Yaskawa INFORM job: pointsclTRJ1.JBI

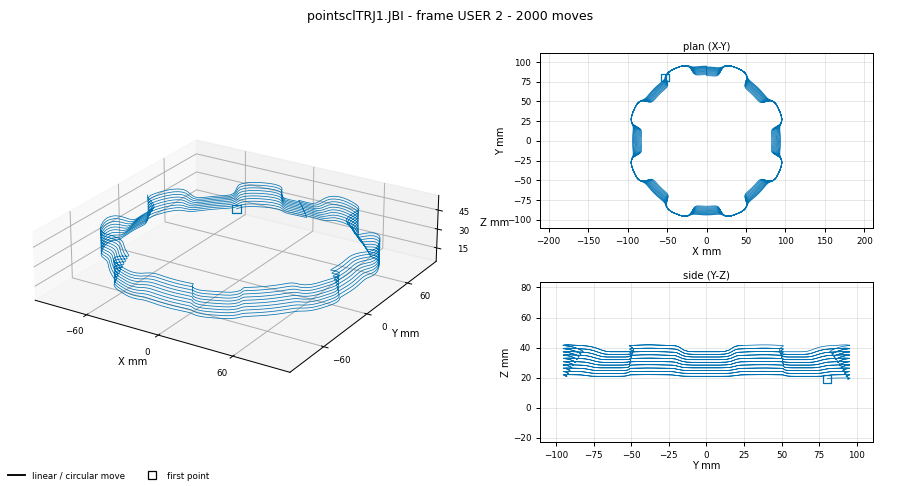
[picture p0: tool path of pointsclTRJ1.JBI in frame USER 2, 2000 of 2000 moves have a stored position in this frame; points joined in program order, loops and branches not executed]
/JOB
//NAME pointsclTRJ1
//POS
///NPOS 2000,0,0,0,0,0
///USER 2
///TOOL 1
///POSTYPE USER
///RECTAN
///RCONF 1,0,0,0,0,0,0,0,0,0,0,0,0,0,0,0,0,0,0,0,0,0,0,0
C00000=-52.755,80.388,19.309,-159.4943,21.2238,0.0000
C00001=-51.961,81.931,19.493,-161.2614,21.3884,0.0000
C00002=-51.163,83.502,19.627,-163.2617,21.3173,0.0000
C00003=-49.917,85.194,19.692,-165.6695,20.6930,0.0000
C00004=-47.874,87.106,19.726,-168.7116,19.3736,0.0000
C00005=-45.272,88.975,19.753,-171.6554,17.3027,0.0000
C00006=-42.449,90.515,19.780,-179.9091,0.0437,0.0000
C00007=-39.659,91.796,19.798,-179.9891,0.0048,0.0000
C00008=-36.867,92.953,19.798,-179.9889,0.0043,0.0000
C00009=-33.988,94.020,19.780,-179.9048,0.0334,0.0000
C00010=-30.903,94.927,19.753,-161.9258,-6.4497,0.0000
C00011=-27.741,95.446,19.726,-158.4611,-5.9689,0.0000
C00012=-24.945,95.538,19.692,-155.4722,-4.9413,0.0000
C00013=-22.867,95.222,19.627,-153.3983,-3.8614,0.0000
C00014=-21.192,94.676,19.493,-151.9726,-2.6572,0.0000
C00015=-19.540,94.146,19.309,-150.8542,-1.4373,0.0000
C00016=-17.528,93.824,19.120,-149.8453,-0.1078,0.0000
C00017=-14.592,93.857,18.976,-148.8983,1.4069,0.0000
C00018=-10.190,94.262,18.917,-148.2538,2.5071,0.0000
C00019=-5.317,94.652,18.914,-148.1214,1.7626,0.0000
C00020=0.000,94.804,18.916,-148.0939,0.0004,0.0000
C00021=0.000,93.772,20.859,-146.9132,0.0004,0.0000
C00022=5.223,93.624,20.857,-146.9416,-1.8172,0.0000
C00023=10.031,93.243,20.860,-147.0713,-2.4820,0.0000
C00024=14.399,92.874,20.935,-147.7018,-1.1471,0.0000
C00025=17.292,92.935,21.118,-148.6350,0.5162,0.0000
C00026=19.271,93.399,21.361,-149.6419,1.9341,0.0000
C00027=20.902,94.108,21.598,-150.7809,3.2271,0.0000
C00028=22.556,94.852,21.773,-152.2300,4.6103,0.0000
C00029=24.607,95.353,21.858,-154.3520,5.8653,0.0000
C00030=27.423,95.407,21.902,-157.4539,7.0484,0.0000
C00031=30.651,94.973,21.938,-161.0071,7.6664,0.0000
C00032=33.828,94.073,21.973,-164.2005,7.6094,0.0000
C00033=36.813,92.974,21.997,-179.9889,-0.0043,0.0000
C00034=39.712,91.773,21.997,-179.9891,-0.0048,0.0000
C00035=42.599,90.440,21.973,-174.1812,-16.5268,0.0000
C00036=45.483,88.829,21.938,-171.8779,-18.8083,0.0000
C00037=48.072,86.854,21.902,-168.7509,-20.8451,0.0000
C00038=50.025,84.825,21.858,-165.4828,-22.1308,0.0000
C00039=51.121,83.020,21.773,-162.8864,-22.6578,0.0000
C00040=51.765,81.324,21.598,-160.7193,-22.6085,0.0000
C00041=52.416,79.670,21.361,-158.8690,-22.3978,0.0000
C00042=53.488,77.942,21.118,-157.0442,-21.9870,0.0000
C00043=55.491,75.854,20.935,-155.1213,-21.3210,0.0000
C00044=58.840,73.026,20.860,-153.6891,-20.6953,0.0000
C00045=62.509,69.895,20.857,-154.0343,-21.2910,0.0000
C00046=66.307,66.307,20.859,-155.2636,-22.7071,0.0000
C00047=69.895,62.509,20.857,-156.5650,-24.0758,0.0000
C00048=73.026,58.840,20.860,-157.1474,-24.4962,0.0000
C00049=75.854,55.491,20.935,-156.7212,-23.0730,0.0000
C00050=77.942,53.488,21.118,-156.3234,-21.2020,0.0000
C00051=79.670,52.416,21.361,-156.1628,-19.4697,0.0000
C00052=81.324,51.765,21.598,-156.1941,-17.7476,0.0000
C00053=83.020,51.121,21.773,-156.4051,-15.7569,0.0000
C00054=84.825,50.025,21.858,-157.2128,-13.4268,0.0000
C00055=86.854,48.072,21.902,-158.7826,-10.5041,0.0000
C00056=88.829,45.483,21.938,-161.0147,-7.6857,0.0000
C00057=90.440,42.599,21.973,-163.3923,-5.5777,0.0000
C00058=91.773,39.712,21.997,-179.9952,-0.0109,0.0000
C00059=92.974,36.813,21.997,-179.9957,-0.0111,0.0000
C00060=94.073,33.828,21.973,172.0955,-15.6567,0.0000
C00061=94.973,30.651,21.938,171.8979,-18.8167,0.0000
C00062=95.407,27.423,21.902,172.3749,-22.3664,0.0000
C00063=95.353,24.607,21.858,173.4988,-25.5041,0.0000
C00064=94.852,22.556,21.773,174.7928,-27.6724,0.0000
C00065=94.108,20.902,21.598,176.3037,-29.1683,0.0000
C00066=93.399,19.271,21.361,177.7589,-30.3389,0.0000
C00067=92.935,17.292,21.118,179.3955,-31.3636,0.0000
C00068=92.874,14.399,20.935,-178.6430,-32.2909,0.0000
C00069=93.243,10.031,20.860,-177.0437,-32.8939,0.0000
C00070=93.624,5.223,20.857,-177.8321,-33.0396,0.0000
C00071=93.772,0.000,20.859,179.9995,-33.0868,0.0000
C00072=93.624,-5.223,20.857,177.8327,-33.0396,0.0000
C00073=93.243,-10.031,20.860,177.0444,-32.8939,0.0000
C00074=92.875,-14.399,20.935,178.6429,-32.2908,0.0000
C00075=92.935,-17.292,21.118,-179.3958,-31.3634,0.0000
C00076=93.399,-19.271,21.361,-177.7592,-30.3389,0.0000
C00077=94.108,-20.902,21.598,-176.3039,-29.1683,0.0000
C00078=94.852,-22.556,21.773,-174.7928,-27.6724,0.0000
C00079=95.353,-24.607,21.858,-173.4988,-25.5041,0.0000
C00080=95.407,-27.423,21.902,-172.3749,-22.3664,0.0000
C00081=94.973,-30.651,21.938,-171.8979,-18.8167,0.0000
C00082=94.073,-33.828,21.973,-172.0955,-15.6567,0.0000
C00083=92.974,-36.813,21.997,179.9957,-0.0111,0.0000
C00084=91.773,-39.712,21.997,179.9952,-0.0109,0.0000
C00085=90.440,-42.599,21.973,163.3923,-5.5777,0.0000
C00086=88.829,-45.483,21.938,161.0147,-7.6857,0.0000
C00087=86.854,-48.072,21.902,158.7826,-10.5041,0.0000
C00088=84.825,-50.025,21.858,157.2128,-13.4268,0.0000
C00089=83.020,-51.121,21.773,156.4050,-15.7569,0.0000
C00090=81.324,-51.765,21.598,156.1939,-17.7474,0.0000
C00091=79.670,-52.416,21.361,156.1625,-19.4695,0.0000
C00092=77.942,-53.488,21.118,156.3231,-21.2019,0.0000
C00093=75.854,-55.491,20.935,156.7211,-23.0731,0.0000
C00094=73.026,-58.840,20.860,157.1478,-24.4967,0.0000
C00095=69.895,-62.509,20.857,156.5653,-24.0762,0.0000
C00096=66.307,-66.307,20.859,155.2630,-22.7065,0.0000
C00097=62.509,-69.895,20.857,154.0346,-21.2914,0.0000
C00098=58.840,-73.026,20.860,153.6895,-20.6957,0.0000
C00099=55.491,-75.854,20.935,155.1214,-21.3209,0.0000
C00100=53.488,-77.942,21.118,157.0440,-21.9867,0.0000
C00101=52.416,-79.670,21.361,158.8689,-22.3975,0.0000
C00102=51.765,-81.324,21.598,160.7192,-22.6084,0.0000
C00103=51.121,-83.020,21.773,162.8864,-22.6578,0.0000
C00104=50.025,-84.825,21.858,165.4828,-22.1308,0.0000
C00105=48.072,-86.854,21.902,168.7509,-20.8451,0.0000
C00106=45.483,-88.829,21.938,171.8779,-18.8083,0.0000
C00107=42.599,-90.440,21.973,174.1812,-16.5268,0.0000
C00108=39.712,-91.773,21.997,179.9891,-0.0048,0.0000
C00109=36.813,-92.974,21.997,179.9889,-0.0043,0.0000
C00110=33.828,-94.073,21.973,164.2005,7.6094,0.0000
C00111=30.651,-94.973,21.938,161.0071,7.6664,0.0000
C00112=27.423,-95.407,21.902,157.4539,7.0484,0.0000
C00113=24.607,-95.353,21.858,154.3520,5.8653,0.0000
C00114=22.556,-94.852,21.773,152.2300,4.6103,0.0000
C00115=20.902,-94.108,21.598,150.7809,3.2271,0.0000
C00116=19.271,-93.399,21.361,149.6419,1.9341,0.0000
C00117=17.292,-92.935,21.118,148.6350,0.5162,0.0000
C00118=14.399,-92.874,20.935,147.7018,-1.1471,0.0000
C00119=10.031,-93.243,20.860,147.0713,-2.4820,0.0000
C00120=5.223,-93.624,20.857,146.9416,-1.8172,0.0000
C00121=0.000,-93.772,20.859,146.9132,0.0004,0.0000
C00122=0.000,-93.772,20.859,146.9132,0.0004,0.0000
C00123=-5.223,-93.624,20.857,146.9416,1.8167,0.0000
C00124=-10.031,-93.243,20.860,147.0713,2.4814,0.0000
C00125=-14.399,-92.875,20.935,147.7020,1.1472,0.0000
C00126=-17.292,-92.935,21.118,148.6351,-0.5159,0.0000
C00127=-19.271,-93.399,21.361,149.6420,-1.9338,0.0000
C00128=-20.902,-94.108,21.598,150.7809,-3.2269,0.0000
C00129=-22.556,-94.852,21.773,152.2300,-4.6102,0.0000
C00130=-24.607,-95.353,21.858,154.3520,-5.8653,0.0000
C00131=-27.423,-95.407,21.902,157.4539,-7.0484,0.0000
C00132=-30.651,-94.973,21.938,161.0071,-7.6664,0.0000
C00133=-33.828,-94.073,21.973,164.2005,-7.6094,0.0000
C00134=-36.813,-92.974,21.997,179.9889,0.0043,0.0000
C00135=-39.712,-91.773,21.997,179.9891,0.0048,0.0000
C00136=-42.599,-90.440,21.973,174.1812,16.5268,0.0000
C00137=-45.483,-88.829,21.938,171.8779,18.8083,0.0000
C00138=-48.072,-86.854,21.902,168.7509,20.8451,0.0000
C00139=-50.025,-84.825,21.858,165.4828,22.1308,0.0000
C00140=-51.121,-83.020,21.773,162.8864,22.6578,0.0000
C00141=-51.765,-81.324,21.598,160.7193,22.6085,0.0000
C00142=-52.416,-79.670,21.361,158.8690,22.3978,0.0000
C00143=-53.488,-77.942,21.118,157.0442,21.9870,0.0000
C00144=-55.491,-75.854,20.935,155.1213,21.3210,0.0000
C00145=-58.840,-73.026,20.860,153.6891,20.6953,0.0000
C00146=-62.509,-69.895,20.857,154.0343,21.2910,0.0000
C00147=-66.307,-66.307,20.859,155.2636,22.7071,0.0000
C00148=-69.895,-62.509,20.857,156.5650,24.0758,0.0000
C00149=-73.026,-58.840,20.860,157.1474,24.4962,0.0000
C00150=-75.854,-55.491,20.935,156.7212,23.0730,0.0000
C00151=-77.942,-53.488,21.118,156.3234,21.2020,0.0000
C00152=-79.670,-52.416,21.361,156.1628,19.4697,0.0000
C00153=-81.324,-51.765,21.598,156.1941,17.7476,0.0000
C00154=-83.020,-51.121,21.773,156.4051,15.7569,0.0000
C00155=-84.825,-50.025,21.858,157.2128,13.4268,0.0000
C00156=-86.854,-48.072,21.902,158.7826,10.5041,0.0000
C00157=-88.829,-45.483,21.938,161.0147,7.6857,0.0000
C00158=-90.440,-42.599,21.973,163.3923,5.5777,0.0000
C00159=-91.773,-39.712,21.997,179.9952,0.0109,0.0000
C00160=-92.974,-36.813,21.997,179.9957,0.0111,0.0000
C00161=-94.073,-33.828,21.973,-172.0955,15.6567,0.0000
C00162=-94.973,-30.651,21.938,-171.8979,18.8167,0.0000
C00163=-95.407,-27.423,21.902,-172.3749,22.3664,0.0000
C00164=-95.353,-24.607,21.858,-173.4988,25.5041,0.0000
C00165=-94.852,-22.556,21.773,-174.7928,27.6724,0.0000
C00166=-94.108,-20.902,21.598,-176.3037,29.1683,0.0000
C00167=-93.399,-19.271,21.361,-177.7589,30.3389,0.0000
C00168=-92.935,-17.292,21.118,-179.3955,31.3636,0.0000
C00169=-92.874,-14.399,20.935,178.6430,32.2909,0.0000
C00170=-93.243,-10.031,20.860,177.0437,32.8939,0.0000
C00171=-93.624,-5.223,20.857,177.8321,33.0396,0.0000
C00172=-93.772,0.000,20.859,-179.9995,33.0868,0.0000
C00173=-93.624,5.223,20.857,-177.8327,33.0396,0.0000
C00174=-93.243,10.031,20.860,-177.0444,32.8939,0.0000
C00175=-92.875,14.399,20.935,-178.6429,32.2908,0.0000
C00176=-92.935,17.292,21.118,179.3958,31.3634,0.0000
C00177=-93.399,19.271,21.361,177.7592,30.3389,0.0000
C00178=-94.108,20.902,21.598,176.3039,29.1683,0.0000
C00179=-94.852,22.556,21.773,174.7928,27.6724,0.0000
C00180=-95.353,24.607,21.858,173.4988,25.5041,0.0000
C00181=-95.407,27.423,21.902,172.3749,22.3664,0.0000
C00182=-94.973,30.651,21.938,171.8979,18.8167,0.0000
C00183=-94.073,33.828,21.973,172.0955,15.6567,0.0000
C00184=-92.974,36.813,21.997,-179.9957,0.0111,0.0000
C00185=-91.773,39.712,21.997,-179.9952,0.0109,0.0000
C00186=-90.440,42.599,21.973,-163.3923,5.5777,0.0000
C00187=-88.829,45.483,21.938,-161.0147,7.6857,0.0000
C00188=-86.854,48.072,21.902,-158.7826,10.5041,0.0000
C00189=-84.825,50.025,21.858,-157.2128,13.4268,0.0000
C00190=-83.020,51.121,21.773,-156.4050,15.7569,0.0000
C00191=-81.324,51.765,21.598,-156.1939,17.7474,0.0000
C00192=-79.670,52.416,21.361,-156.1625,19.4695,0.0000
C00193=-77.942,53.488,21.118,-156.3231,21.2019,0.0000
C00194=-75.854,55.491,20.935,-156.7211,23.0731,0.0000
C00195=-73.026,58.840,20.860,-157.1478,24.4967,0.0000
C00196=-69.895,62.509,20.857,-156.5653,24.0762,0.0000
C00197=-66.307,66.307,20.859,-155.2630,22.7065,0.0000
C00198=-62.509,69.895,20.857,-154.0346,21.2914,0.0000
C00199=-58.840,73.026,20.860,-153.6895,20.6957,0.0000
C00200=-55.491,75.854,20.935,-155.1214,21.3209,0.0000
C00201=-53.488,77.942,21.118,-157.0440,21.9867,0.0000
C00202=-52.416,79.670,21.361,-158.8689,22.3975,0.0000
C00203=-51.765,81.324,21.598,-160.7192,22.6084,0.0000
C00204=-51.121,83.020,21.773,-162.8864,22.6578,0.0000
C00205=-50.025,84.825,21.858,-165.4828,22.1308,0.0000
C00206=-48.072,86.854,21.902,-168.7509,20.8451,0.0000
C00207=-45.483,88.829,21.938,-171.8779,18.8083,0.0000
C00208=-42.599,90.440,21.973,-174.1812,16.5268,0.0000
C00209=-39.712,91.773,21.997,-179.9891,0.0048,0.0000
C00210=-36.813,92.974,21.997,-179.9889,0.0043,0.0000
C00211=-33.828,94.073,21.973,-164.2005,-7.6094,0.0000
C00212=-30.651,94.973,21.938,-161.0071,-7.6664,0.0000
C00213=-27.423,95.407,21.902,-157.4539,-7.0484,0.0000
C00214=-24.607,95.353,21.858,-154.3520,-5.8653,0.0000
C00215=-22.556,94.852,21.773,-152.2300,-4.6102,0.0000
C00216=-20.902,94.108,21.598,-150.7809,-3.2269,0.0000
C00217=-19.271,93.399,21.361,-149.6420,-1.9338,0.0000
C00218=-17.292,92.935,21.118,-148.6351,-0.5159,0.0000
C00219=-14.399,92.875,20.935,-147.7020,1.1472,0.0000
C00220=-10.031,93.243,20.860,-147.0713,2.4814,0.0000
C00221=-5.223,93.624,20.857,-146.9416,1.8167,0.0000
C00222=0.000,93.772,20.859,-146.9132,0.0004,0.0000
C00223=0.000,92.684,22.771,-145.8888,0.0004,0.0000
C00224=5.124,92.540,22.769,-145.9181,-1.8620,0.0000
C00225=9.864,92.169,22.773,-146.0452,-2.4396,0.0000
C00226=14.194,91.838,22.865,-146.6687,-0.8798,0.0000
C00227=17.042,91.994,23.091,-147.5969,0.9153,0.0000
C00228=18.986,92.606,23.393,-148.6082,2.4100,0.0000
C00229=20.592,93.503,23.691,-149.7732,3.7684,0.0000
C00230=22.223,94.456,23.912,-151.2813,5.2238,0.0000
C00231=24.245,95.156,24.019,-153.4766,6.7389,0.0000
C00232=27.082,95.366,24.075,-156.7610,8.0545,0.0000
C00233=30.380,95.022,24.120,-160.5087,8.7471,0.0000
C00234=33.658,94.129,24.166,-163.7677,8.7396,0.0000
C00235=36.755,92.996,24.196,-179.9893,-0.0042,0.0000
C00236=39.769,91.748,24.196,-179.9895,-0.0046,0.0000
C00237=42.760,90.359,24.166,-174.7067,-17.6262,0.0000
C00238=45.709,88.673,24.120,-172.3190,-19.9210,0.0000
C00239=48.284,86.584,24.075,-168.9803,-22.0444,0.0000
C00240=50.142,84.429,24.019,-165.4510,-23.3634,0.0000
C00241=51.076,82.504,23.912,-162.5826,-23.7496,0.0000
C00242=51.556,80.678,23.691,-160.2983,-23.6832,0.0000
C00243=52.057,78.907,23.393,-158.3658,-23.4364,0.0000
C00244=52.999,77.101,23.091,-156.4709,-22.9648,0.0000
C00245=54.903,74.976,22.865,-154.4508,-22.1874,0.0000
C00246=58.198,72.148,22.773,-152.8667,-21.3762,0.0000
C00247=61.813,69.059,22.769,-153.1525,-21.9046,0.0000
C00248=65.538,65.538,22.771,-154.4083,-23.3627,0.0000
C00249=69.059,61.813,22.769,-155.7401,-24.7719,0.0000
C00250=72.148,58.198,22.773,-156.2588,-25.1304,0.0000
C00251=74.976,54.903,22.865,-155.6753,-23.5376,0.0000
C00252=77.101,52.999,23.091,-155.1950,-21.5663,0.0000
C00253=78.907,52.057,23.393,-154.9986,-19.7713,0.0000
C00254=80.678,51.556,23.691,-155.0197,-17.9829,0.0000
C00255=82.504,51.076,23.912,-155.2435,-15.9014,0.0000
C00256=84.429,50.142,24.019,-155.9492,-13.3330,0.0000
C00257=86.584,48.284,24.075,-157.5822,-10.2051,0.0000
C00258=88.673,45.709,24.120,-159.9130,-7.2188,0.0000
C00259=90.359,42.760,24.166,-162.3030,-5.0442,0.0000
C00260=91.748,39.769,24.196,-179.9954,-0.0105,0.0000
C00261=92.996,36.755,24.196,-179.9958,-0.0107,0.0000
C00262=94.129,33.658,24.166,170.9035,-16.0387,0.0000
C00263=95.022,30.380,24.120,170.7301,-19.2556,0.0000
C00264=95.366,27.082,24.075,171.2449,-22.9965,0.0000
C00265=95.156,24.245,24.019,172.4771,-26.3260,0.0000
C00266=94.456,22.223,23.912,174.0484,-28.5884,0.0000
C00267=93.503,20.592,23.691,175.6407,-30.1546,0.0000
C00268=92.606,18.986,23.393,177.1774,-31.3609,0.0000
C00269=91.994,17.042,23.091,178.9159,-32.3984,0.0000
C00270=91.838,14.194,22.865,-178.9471,-33.3268,0.0000
C00271=92.169,9.864,22.773,-177.0596,-33.9199,0.0000
C00272=92.540,5.124,22.769,-177.7522,-34.0614,0.0000
C00273=92.684,0.000,22.771,179.9995,-34.1112,0.0000
C00274=92.540,-5.124,22.769,177.7528,-34.0615,0.0000
C00275=92.169,-9.864,22.773,177.0604,-33.9198,0.0000
C00276=91.838,-14.194,22.865,178.9470,-33.3267,0.0000
C00277=91.994,-17.042,23.091,-178.9163,-32.3983,0.0000
C00278=92.606,-18.986,23.393,-177.1778,-31.3608,0.0000
C00279=93.503,-20.592,23.691,-175.6410,-30.1546,0.0000
C00280=94.456,-22.223,23.912,-174.0485,-28.5884,0.0000
C00281=95.156,-24.245,24.019,-172.4771,-26.3260,0.0000
C00282=95.366,-27.082,24.075,-171.2449,-22.9965,0.0000
C00283=95.022,-30.380,24.120,-170.7301,-19.2556,0.0000
C00284=94.129,-33.658,24.166,-170.9035,-16.0387,0.0000
C00285=92.996,-36.755,24.196,179.9958,-0.0107,0.0000
C00286=91.748,-39.769,24.196,179.9954,-0.0105,0.0000
C00287=90.359,-42.760,24.166,162.3030,-5.0442,0.0000
C00288=88.673,-45.709,24.120,159.9130,-7.2188,0.0000
C00289=86.584,-48.284,24.075,157.5822,-10.2051,0.0000
C00290=84.429,-50.142,24.019,155.9492,-13.3330,0.0000
C00291=82.504,-51.076,23.912,155.2435,-15.9013,0.0000
C00292=80.678,-51.556,23.691,155.0196,-17.9828,0.0000
C00293=78.907,-52.057,23.393,154.9983,-19.7711,0.0000
C00294=77.101,-52.999,23.091,155.1947,-21.5661,0.0000
C00295=74.976,-54.903,22.865,155.6752,-23.5376,0.0000
C00296=72.148,-58.198,22.773,156.2592,-25.1309,0.0000
C00297=69.059,-61.813,22.769,155.7405,-24.7723,0.0000
C00298=65.538,-65.538,22.771,154.4077,-23.3621,0.0000
C00299=61.813,-69.059,22.769,153.1528,-21.9050,0.0000
C00300=58.198,-72.148,22.773,152.8672,-21.3767,0.0000
C00301=54.903,-74.976,22.865,154.4508,-22.1873,0.0000
C00302=52.999,-77.101,23.091,156.4708,-22.9645,0.0000
C00303=52.057,-78.907,23.393,158.3656,-23.4361,0.0000
C00304=51.556,-80.678,23.691,160.2982,-23.6830,0.0000
C00305=51.076,-82.504,23.912,162.5826,-23.7495,0.0000
C00306=50.142,-84.429,24.019,165.4510,-23.3634,0.0000
C00307=48.284,-86.584,24.075,168.9803,-22.0444,0.0000
C00308=45.709,-88.673,24.120,172.3190,-19.9210,0.0000
C00309=42.760,-90.359,24.166,174.7067,-17.6262,0.0000
C00310=39.769,-91.748,24.196,179.9895,-0.0046,0.0000
C00311=36.755,-92.996,24.196,179.9893,-0.0042,0.0000
C00312=33.658,-94.129,24.166,163.7677,8.7396,0.0000
C00313=30.380,-95.022,24.120,160.5087,8.7471,0.0000
C00314=27.082,-95.366,24.075,156.7610,8.0545,0.0000
C00315=24.245,-95.156,24.019,153.4766,6.7389,0.0000
C00316=22.223,-94.456,23.912,151.2813,5.2238,0.0000
C00317=20.592,-93.503,23.691,149.7732,3.7684,0.0000
C00318=18.986,-92.606,23.393,148.6082,2.4100,0.0000
C00319=17.042,-91.994,23.091,147.5969,0.9153,0.0000
C00320=14.194,-91.838,22.865,146.6687,-0.8798,0.0000
C00321=9.864,-92.169,22.773,146.0452,-2.4396,0.0000
C00322=5.124,-92.540,22.769,145.9181,-1.8620,0.0000
C00323=0.000,-92.684,22.771,145.8888,0.0004,0.0000
C00324=0.000,-92.684,22.771,145.8888,0.0004,0.0000
C00325=-5.124,-92.540,22.769,145.9181,1.8615,0.0000
C00326=-9.864,-92.169,22.773,146.0452,2.4390,0.0000
C00327=-14.194,-91.838,22.865,146.6688,0.8798,0.0000
C00328=-17.042,-91.994,23.091,147.5970,-0.9150,0.0000
C00329=-18.986,-92.606,23.393,148.6082,-2.4097,0.0000
C00330=-20.592,-93.503,23.691,149.7733,-3.7682,0.0000
C00331=-22.223,-94.456,23.912,151.2813,-5.2237,0.0000
C00332=-24.245,-95.156,24.019,153.4766,-6.7389,0.0000
C00333=-27.082,-95.366,24.075,156.7610,-8.0545,0.0000
C00334=-30.380,-95.022,24.120,160.5087,-8.7471,0.0000
C00335=-33.658,-94.129,24.166,163.7677,-8.7396,0.0000
C00336=-36.755,-92.996,24.196,179.9893,0.0042,0.0000
C00337=-39.769,-91.748,24.196,179.9895,0.0046,0.0000
C00338=-42.760,-90.359,24.166,174.7067,17.6262,0.0000
C00339=-45.709,-88.673,24.120,172.3190,19.9210,0.0000
C00340=-48.284,-86.584,24.075,168.9803,22.0444,0.0000
C00341=-50.142,-84.429,24.019,165.4510,23.3634,0.0000
C00342=-51.076,-82.504,23.912,162.5826,23.7496,0.0000
C00343=-51.556,-80.678,23.691,160.2983,23.6832,0.0000
C00344=-52.057,-78.907,23.393,158.3658,23.4364,0.0000
C00345=-52.999,-77.101,23.091,156.4709,22.9648,0.0000
C00346=-54.903,-74.976,22.865,154.4508,22.1874,0.0000
C00347=-58.198,-72.148,22.773,152.8667,21.3762,0.0000
C00348=-61.813,-69.059,22.769,153.1525,21.9046,0.0000
C00349=-65.538,-65.538,22.771,154.4083,23.3627,0.0000
C00350=-69.059,-61.813,22.769,155.7401,24.7719,0.0000
C00351=-72.148,-58.198,22.773,156.2588,25.1304,0.0000
C00352=-74.976,-54.903,22.865,155.6753,23.5376,0.0000
C00353=-77.101,-52.999,23.091,155.1950,21.5663,0.0000
C00354=-78.907,-52.057,23.393,154.9986,19.7713,0.0000
C00355=-80.678,-51.556,23.691,155.0197,17.9829,0.0000
C00356=-82.504,-51.076,23.912,155.2435,15.9014,0.0000
C00357=-84.429,-50.142,24.019,155.9492,13.3330,0.0000
C00358=-86.584,-48.284,24.075,157.5822,10.2051,0.0000
C00359=-88.673,-45.709,24.120,159.9130,7.2188,0.0000
C00360=-90.359,-42.760,24.166,162.3030,5.0442,0.0000
C00361=-91.748,-39.769,24.196,179.9954,0.0105,0.0000
C00362=-92.996,-36.755,24.196,179.9958,0.0107,0.0000
C00363=-94.129,-33.658,24.166,-170.9035,16.0387,0.0000
C00364=-95.022,-30.380,24.120,-170.7301,19.2556,0.0000
C00365=-95.366,-27.082,24.075,-171.2449,22.9965,0.0000
C00366=-95.156,-24.245,24.019,-172.4771,26.3260,0.0000
C00367=-94.456,-22.223,23.912,-174.0484,28.5884,0.0000
C00368=-93.503,-20.592,23.691,-175.6407,30.1546,0.0000
C00369=-92.606,-18.986,23.393,-177.1774,31.3609,0.0000
C00370=-91.994,-17.042,23.091,-178.9159,32.3984,0.0000
C00371=-91.838,-14.194,22.865,178.9471,33.3268,0.0000
C00372=-92.169,-9.864,22.773,177.0596,33.9199,0.0000
C00373=-92.540,-5.124,22.769,177.7522,34.0614,0.0000
C00374=-92.684,0.000,22.771,-179.9995,34.1112,0.0000
C00375=-92.540,5.124,22.769,-177.7528,34.0615,0.0000
C00376=-92.169,9.864,22.773,-177.0604,33.9198,0.0000
C00377=-91.838,14.194,22.865,-178.9470,33.3267,0.0000
C00378=-91.994,17.042,23.091,178.9163,32.3983,0.0000
C00379=-92.606,18.986,23.393,177.1778,31.3608,0.0000
C00380=-93.503,20.592,23.691,175.6410,30.1546,0.0000
C00381=-94.456,22.223,23.912,174.0485,28.5884,0.0000
C00382=-95.156,24.245,24.019,172.4771,26.3260,0.0000
C00383=-95.366,27.082,24.075,171.2449,22.9965,0.0000
C00384=-95.022,30.380,24.120,170.7301,19.2556,0.0000
C00385=-94.129,33.658,24.166,170.9035,16.0387,0.0000
C00386=-92.996,36.755,24.196,-179.9958,0.0107,0.0000
C00387=-91.748,39.769,24.196,-179.9954,0.0105,0.0000
C00388=-90.359,42.760,24.166,-162.3030,5.0442,0.0000
C00389=-88.673,45.709,24.120,-159.9130,7.2188,0.0000
C00390=-86.584,48.284,24.075,-157.5822,10.2051,0.0000
C00391=-84.429,50.142,24.019,-155.9492,13.3330,0.0000
C00392=-82.504,51.076,23.912,-155.2435,15.9013,0.0000
C00393=-80.678,51.556,23.691,-155.0196,17.9828,0.0000
C00394=-78.907,52.057,23.393,-154.9983,19.7711,0.0000
C00395=-77.101,52.999,23.091,-155.1947,21.5661,0.0000
C00396=-74.976,54.903,22.865,-155.6752,23.5376,0.0000
C00397=-72.148,58.198,22.773,-156.2592,25.1309,0.0000
C00398=-69.059,61.813,22.769,-155.7405,24.7723,0.0000
C00399=-65.538,65.538,22.771,-154.4077,23.3621,0.0000
C00400=-61.813,69.059,22.769,-153.1528,21.9050,0.0000
C00401=-58.198,72.148,22.773,-152.8672,21.3767,0.0000
C00402=-54.903,74.976,22.865,-154.4508,22.1873,0.0000
C00403=-52.999,77.101,23.091,-156.4708,22.9645,0.0000
C00404=-52.057,78.907,23.393,-158.3656,23.4361,0.0000
C00405=-51.556,80.678,23.691,-160.2982,23.6830,0.0000
C00406=-51.076,82.504,23.912,-162.5826,23.7495,0.0000
C00407=-50.142,84.429,24.019,-165.4510,23.3634,0.0000
C00408=-48.284,86.584,24.075,-168.9803,22.0444,0.0000
C00409=-45.709,88.673,24.120,-172.3190,19.9210,0.0000
C00410=-42.760,90.359,24.166,-174.7067,17.6262,0.0000
C00411=-39.769,91.748,24.196,-179.9895,0.0046,0.0000
C00412=-36.755,92.996,24.196,-179.9893,0.0042,0.0000
C00413=-33.658,94.129,24.166,-163.7677,-8.7396,0.0000
C00414=-30.380,95.022,24.120,-160.5087,-8.7471,0.0000
C00415=-27.082,95.366,24.075,-156.7610,-8.0545,0.0000
C00416=-24.245,95.156,24.019,-153.4766,-6.7389,0.0000
C00417=-22.223,94.456,23.912,-151.2813,-5.2237,0.0000
C00418=-20.592,93.503,23.691,-149.7733,-3.7682,0.0000
C00419=-18.986,92.606,23.393,-148.6082,-2.4097,0.0000
C00420=-17.042,91.994,23.091,-147.5970,-0.9150,0.0000
C00421=-14.194,91.838,22.865,-146.6688,0.8798,0.0000
C00422=-9.864,92.169,22.773,-146.0452,2.4390,0.0000
C00423=-5.124,92.540,22.769,-145.9181,1.8615,0.0000
C00424=0.000,92.684,22.771,-145.8888,0.0004,0.0000
C00425=0.000,91.548,24.655,-144.9980,0.0004,0.0000
C00426=5.020,91.408,24.652,-145.0279,-1.8988,0.0000
C00427=9.690,91.047,24.657,-145.1527,-2.3842,0.0000
C00428=13.981,90.755,24.767,-145.7748,-0.6100,0.0000
C00429=16.781,91.008,25.041,-146.7039,1.3008,0.0000
C00430=18.686,91.772,25.406,-147.7228,2.8612,0.0000
C00431=20.265,92.865,25.771,-148.9167,4.2814,0.0000
C00432=21.871,94.037,26.043,-150.4888,5.8096,0.0000
C00433=23.861,94.948,26.175,-152.7985,7.5672,0.0000
C00434=26.720,95.323,26.245,-156.3222,8.9978,0.0000
C00435=30.093,95.074,26.301,-160.3364,9.7146,0.0000
C00436=33.476,94.189,26.358,-163.7368,9.6720,0.0000
C00437=36.693,93.020,26.395,-179.9900,-0.0039,0.0000
C00438=39.829,91.721,26.395,-179.9902,-0.0043,0.0000
C00439=42.931,90.273,26.358,-175.3837,-18.3011,0.0000
C00440=45.948,88.507,26.301,-172.9244,-20.7227,0.0000
C00441=48.509,86.297,26.245,-169.3630,-23.0207,0.0000
C00442=50.266,84.010,26.175,-165.5434,-24.4272,0.0000
C00443=51.029,81.959,26.043,-162.3815,-24.7149,0.0000
C00444=51.336,79.995,25.771,-159.9751,-24.6351,0.0000
C00445=51.679,78.105,25.406,-157.9609,-24.3577,0.0000
C00446=52.487,76.218,25.041,-156.0012,-23.8366,0.0000
C00447=54.287,74.059,24.767,-153.8902,-22.9644,0.0000
C00448=57.528,71.231,24.657,-152.1573,-21.9792,0.0000
C00449=61.085,68.184,24.652,-152.3807,-22.4356,0.0000
C00450=64.734,64.734,24.655,-153.6576,-23.9291,0.0000
C00451=68.184,61.085,24.652,-155.0141,-25.3724,0.0000
C00452=71.231,57.528,24.657,-155.4655,-25.6639,0.0000
C00453=74.059,54.287,24.767,-154.7375,-23.9045,0.0000
C00454=76.218,52.487,25.041,-154.1908,-21.8407,0.0000
C00455=78.105,51.679,25.406,-153.9685,-19.9892,0.0000
C00456=79.995,51.336,25.771,-153.9839,-18.1354,0.0000
C00457=81.959,51.029,26.043,-154.2235,-15.9593,0.0000
C00458=84.010,50.266,26.175,-154.8713,-13.1382,0.0000
C00459=86.297,48.509,26.245,-156.6197,-9.7812,0.0000
C00460=88.507,45.948,26.301,-159.1319,-6.6157,0.0000
C00461=90.273,42.931,26.358,-161.6434,-4.3823,0.0000
C00462=91.721,39.829,26.395,-179.9957,-0.0098,0.0000
C00463=93.020,36.693,26.395,-179.9961,-0.0100,0.0000
C00464=94.189,33.476,26.358,169.9329,-16.0258,0.0000
C00465=95.074,30.093,26.301,169.6963,-19.3703,0.0000
C00466=95.323,26.720,26.245,170.1905,-23.3690,0.0000
C00467=94.948,23.861,26.175,171.5048,-26.9454,0.0000
C00468=94.037,21.871,26.043,173.3316,-29.3448,0.0000
C00469=92.865,20.265,25.771,175.0042,-30.9870,0.0000
C00470=91.772,18.686,25.406,176.6170,-32.2321,0.0000
C00471=91.008,16.781,25.041,178.4438,-33.2864,0.0000
C00472=90.755,13.981,24.767,-179.2623,-34.2230,0.0000
C00473=91.047,9.690,24.657,-177.0956,-34.8128,0.0000
C00474=91.408,5.020,24.652,-177.6831,-34.9501,0.0000
C00475=91.548,0.000,24.655,179.9995,-35.0020,0.0000
C00476=91.408,-5.020,24.652,177.6838,-34.9501,0.0000
C00477=91.047,-9.690,24.657,177.0965,-34.8128,0.0000
C00478=90.755,-13.981,24.767,179.2623,-34.2228,0.0000
C00479=91.008,-16.781,25.041,-178.4442,-33.2863,0.0000
C00480=91.772,-18.686,25.406,-176.6174,-32.2320,0.0000
C00481=92.865,-20.265,25.771,-175.0045,-30.9870,0.0000
C00482=94.037,-21.871,26.043,-173.3318,-29.3448,0.0000
C00483=94.948,-23.861,26.175,-171.5048,-26.9454,0.0000
C00484=95.323,-26.720,26.245,-170.1905,-23.3690,0.0000
C00485=95.074,-30.093,26.301,-169.6963,-19.3703,0.0000
C00486=94.189,-33.476,26.358,-169.9330,-16.0258,0.0000
C00487=93.020,-36.693,26.395,179.9961,-0.0100,0.0000
C00488=91.721,-39.829,26.395,179.9957,-0.0098,0.0000
C00489=90.273,-42.931,26.358,161.6434,-4.3823,0.0000
C00490=88.507,-45.948,26.301,159.1319,-6.6157,0.0000
C00491=86.297,-48.509,26.245,156.6197,-9.7812,0.0000
C00492=84.010,-50.266,26.175,154.8713,-13.1382,0.0000
C00493=81.959,-51.029,26.043,154.2234,-15.9592,0.0000
C00494=79.995,-51.336,25.771,153.9837,-18.1352,0.0000
C00495=78.105,-51.679,25.406,153.9682,-19.9889,0.0000
C00496=76.218,-52.487,25.041,154.1905,-21.8406,0.0000
C00497=74.059,-54.287,24.767,154.7374,-23.9046,0.0000
C00498=71.231,-57.528,24.657,155.4660,-25.6645,0.0000
C00499=68.184,-61.085,24.652,155.0145,-25.3727,0.0000
C00500=64.734,-64.734,24.655,153.6570,-23.9284,0.0000
C00501=61.085,-68.184,24.652,152.3810,-22.4360,0.0000
C00502=57.528,-71.231,24.657,152.1578,-21.9797,0.0000
C00503=54.287,-74.059,24.767,153.8903,-22.9644,0.0000
C00504=52.487,-76.218,25.041,156.0011,-23.8364,0.0000
C00505=51.679,-78.105,25.406,157.9607,-24.3574,0.0000
C00506=51.336,-79.995,25.771,159.9749,-24.6349,0.0000
C00507=51.029,-81.959,26.043,162.3814,-24.7147,0.0000
C00508=50.266,-84.010,26.175,165.5434,-24.4272,0.0000
C00509=48.509,-86.297,26.245,169.3630,-23.0207,0.0000
C00510=45.948,-88.507,26.301,172.9244,-20.7227,0.0000
C00511=42.931,-90.273,26.358,175.3837,-18.3011,0.0000
C00512=39.829,-91.721,26.395,179.9902,-0.0043,0.0000
C00513=36.693,-93.020,26.395,179.9900,-0.0039,0.0000
C00514=33.476,-94.189,26.358,163.7368,9.6720,0.0000
C00515=30.093,-95.074,26.301,160.3364,9.7146,0.0000
C00516=26.720,-95.323,26.245,156.3222,8.9978,0.0000
C00517=23.861,-94.948,26.175,152.7985,7.5672,0.0000
C00518=21.871,-94.037,26.043,150.4888,5.8096,0.0000
C00519=20.265,-92.865,25.771,148.9167,4.2814,0.0000
C00520=18.686,-91.772,25.406,147.7228,2.8612,0.0000
C00521=16.781,-91.008,25.041,146.7039,1.3008,0.0000
C00522=13.981,-90.755,24.767,145.7748,-0.6100,0.0000
C00523=9.690,-91.047,24.657,145.1527,-2.3842,0.0000
C00524=5.020,-91.408,24.652,145.0279,-1.8988,0.0000
C00525=0.000,-91.548,24.655,144.9980,0.0004,0.0000
C00526=0.000,-91.548,24.655,144.9980,0.0004,0.0000
C00527=-5.020,-91.408,24.652,145.0279,1.8983,0.0000
C00528=-9.690,-91.047,24.657,145.1527,2.3835,0.0000
C00529=-13.981,-90.755,24.767,145.7750,0.6100,0.0000
C00530=-16.781,-91.008,25.041,146.7040,-1.3005,0.0000
C00531=-18.686,-91.772,25.406,147.7229,-2.8609,0.0000
C00532=-20.265,-92.865,25.771,148.9167,-4.2811,0.0000
C00533=-21.871,-94.037,26.043,150.4888,-5.8094,0.0000
C00534=-23.861,-94.948,26.175,152.7985,-7.5672,0.0000
C00535=-26.720,-95.323,26.245,156.3222,-8.9978,0.0000
C00536=-30.093,-95.074,26.301,160.3364,-9.7146,0.0000
C00537=-33.476,-94.189,26.358,163.7368,-9.6720,0.0000
C00538=-36.693,-93.020,26.395,179.9900,0.0039,0.0000
C00539=-39.829,-91.721,26.395,179.9902,0.0043,0.0000
C00540=-42.931,-90.273,26.358,175.3837,18.3011,0.0000
C00541=-45.948,-88.507,26.301,172.9244,20.7227,0.0000
C00542=-48.509,-86.297,26.245,169.3630,23.0207,0.0000
C00543=-50.266,-84.010,26.175,165.5434,24.4272,0.0000
C00544=-51.029,-81.959,26.043,162.3815,24.7149,0.0000
C00545=-51.336,-79.995,25.771,159.9751,24.6351,0.0000
C00546=-51.679,-78.105,25.406,157.9609,24.3577,0.0000
C00547=-52.487,-76.218,25.041,156.0012,23.8366,0.0000
C00548=-54.287,-74.059,24.767,153.8902,22.9644,0.0000
C00549=-57.528,-71.231,24.657,152.1573,21.9792,0.0000
C00550=-61.085,-68.184,24.652,152.3807,22.4356,0.0000
C00551=-64.734,-64.734,24.655,153.6576,23.9291,0.0000
C00552=-68.184,-61.085,24.652,155.0141,25.3724,0.0000
C00553=-71.231,-57.528,24.657,155.4655,25.6639,0.0000
C00554=-74.059,-54.287,24.767,154.7375,23.9045,0.0000
C00555=-76.218,-52.487,25.041,154.1908,21.8407,0.0000
C00556=-78.105,-51.679,25.406,153.9685,19.9892,0.0000
C00557=-79.995,-51.336,25.771,153.9839,18.1354,0.0000
C00558=-81.959,-51.029,26.043,154.2235,15.9593,0.0000
C00559=-84.010,-50.266,26.175,154.8713,13.1382,0.0000
C00560=-86.297,-48.509,26.245,156.6197,9.7812,0.0000
C00561=-88.507,-45.948,26.301,159.1319,6.6157,0.0000
C00562=-90.273,-42.931,26.358,161.6434,4.3823,0.0000
C00563=-91.721,-39.829,26.395,179.9957,0.0098,0.0000
C00564=-93.020,-36.693,26.395,179.9961,0.0100,0.0000
C00565=-94.189,-33.476,26.358,-169.9330,16.0258,0.0000
C00566=-95.074,-30.093,26.301,-169.6963,19.3703,0.0000
C00567=-95.323,-26.720,26.245,-170.1905,23.3690,0.0000
C00568=-94.948,-23.861,26.175,-171.5048,26.9454,0.0000
C00569=-94.037,-21.871,26.043,-173.3316,29.3448,0.0000
C00570=-92.865,-20.265,25.771,-175.0042,30.9870,0.0000
C00571=-91.772,-18.686,25.406,-176.6170,32.2321,0.0000
C00572=-91.008,-16.781,25.041,-178.4438,33.2864,0.0000
C00573=-90.755,-13.981,24.767,179.2623,34.2230,0.0000
C00574=-91.047,-9.690,24.657,177.0956,34.8128,0.0000
C00575=-91.408,-5.020,24.652,177.6831,34.9501,0.0000
C00576=-91.548,0.000,24.655,-179.9995,35.0020,0.0000
C00577=-91.408,5.020,24.652,-177.6838,34.9501,0.0000
C00578=-91.047,9.690,24.657,-177.0965,34.8128,0.0000
C00579=-90.755,13.981,24.767,-179.2623,34.2228,0.0000
C00580=-91.008,16.781,25.041,178.4442,33.2863,0.0000
C00581=-91.772,18.686,25.406,176.6174,32.2320,0.0000
C00582=-92.865,20.265,25.771,175.0045,30.9870,0.0000
C00583=-94.037,21.871,26.043,173.3318,29.3448,0.0000
C00584=-94.948,23.861,26.175,171.5048,26.9454,0.0000
C00585=-95.323,26.720,26.245,170.1905,23.3690,0.0000
C00586=-95.074,30.093,26.301,169.6963,19.3703,0.0000
C00587=-94.189,33.476,26.358,169.9330,16.0258,0.0000
C00588=-93.020,36.693,26.395,-179.9961,0.0100,0.0000
C00589=-91.721,39.829,26.395,-179.9957,0.0098,0.0000
C00590=-90.273,42.931,26.358,-161.6434,4.3823,0.0000
C00591=-88.507,45.948,26.301,-159.1319,6.6157,0.0000
C00592=-86.297,48.509,26.245,-156.6197,9.7812,0.0000
C00593=-84.010,50.266,26.175,-154.8713,13.1382,0.0000
C00594=-81.959,51.029,26.043,-154.2234,15.9592,0.0000
C00595=-79.995,51.336,25.771,-153.9837,18.1352,0.0000
C00596=-78.105,51.679,25.406,-153.9682,19.9889,0.0000
C00597=-76.218,52.487,25.041,-154.1905,21.8406,0.0000
C00598=-74.059,54.287,24.767,-154.7374,23.9046,0.0000
C00599=-71.231,57.528,24.657,-155.4660,25.6645,0.0000
C00600=-68.184,61.085,24.652,-155.0145,25.3727,0.0000
C00601=-64.734,64.734,24.655,-153.6570,23.9284,0.0000
C00602=-61.085,68.184,24.652,-152.3810,22.4360,0.0000
C00603=-57.528,71.231,24.657,-152.1578,21.9797,0.0000
C00604=-54.287,74.059,24.767,-153.8903,22.9644,0.0000
C00605=-52.487,76.218,25.041,-156.0011,23.8364,0.0000
C00606=-51.679,78.105,25.406,-157.9607,24.3574,0.0000
C00607=-51.336,79.995,25.771,-159.9749,24.6349,0.0000
C00608=-51.029,81.959,26.043,-162.3814,24.7147,0.0000
C00609=-50.266,84.010,26.175,-165.5434,24.4272,0.0000
C00610=-48.509,86.297,26.245,-169.3630,23.0207,0.0000
C00611=-45.948,88.507,26.301,-172.9244,20.7227,0.0000
C00612=-42.931,90.273,26.358,-175.3837,18.3011,0.0000
C00613=-39.829,91.721,26.395,-179.9902,0.0043,0.0000
C00614=-36.693,93.020,26.395,-179.9900,0.0039,0.0000
C00615=-33.476,94.189,26.358,-163.7368,-9.6720,0.0000
C00616=-30.093,95.074,26.301,-160.3364,-9.7146,0.0000
C00617=-26.720,95.323,26.245,-156.3222,-8.9978,0.0000
C00618=-23.861,94.948,26.175,-152.7985,-7.5672,0.0000
C00619=-21.871,94.037,26.043,-150.4888,-5.8094,0.0000
C00620=-20.265,92.865,25.771,-148.9167,-4.2811,0.0000
C00621=-18.686,91.772,25.406,-147.7229,-2.8609,0.0000
C00622=-16.781,91.008,25.041,-146.7040,-1.3005,0.0000
C00623=-13.981,90.755,24.767,-145.7750,0.6100,0.0000
C00624=-9.690,91.047,24.657,-145.1527,2.3835,0.0000
C00625=-5.020,91.408,24.652,-145.0279,1.8983,0.0000
C00626=0.000,91.548,24.655,-144.9980,0.0004,0.0000
C00627=0.000,90.369,26.513,-144.2229,0.0004,0.0000
C00628=4.912,90.233,26.509,-144.2533,-1.9288,0.0000
C00629=9.508,89.882,26.515,-144.3761,-2.3187,0.0000
C00630=13.759,89.629,26.645,-145.0013,-0.3412,0.0000
C00631=16.509,89.983,26.968,-145.9347,1.6696,0.0000
C00632=18.373,90.901,27.402,-146.9628,3.2856,0.0000
C00633=19.923,92.196,27.838,-148.1868,4.7664,0.0000
C00634=21.502,93.597,28.166,-149.8272,6.3665,0.0000
C00635=23.458,94.728,28.327,-152.2788,8.3021,0.0000
C00636=26.340,95.277,28.411,-156.1013,9.8857,0.0000
C00637=29.791,95.129,28.479,-160.4391,10.5773,0.0000
C00638=33.285,94.252,28.548,-164.0148,10.4347,0.0000
C00639=36.628,93.045,28.594,-179.9910,-0.0035,0.0000
C00640=39.893,91.693,28.594,-179.9912,-0.0039,0.0000
C00641=43.110,90.182,28.548,-176.1610,-18.6373,0.0000
C00642=46.201,88.332,28.479,-173.6595,-21.2551,0.0000
C00643=48.746,85.996,28.411,-169.8768,-23.8040,0.0000
C00644=50.396,83.570,28.327,-165.6938,-25.3139,0.0000
C00645=50.979,81.387,28.166,-162.2638,-25.5702,0.0000
C00646=51.105,79.281,27.838,-159.7325,-25.4815,0.0000
C00647=51.285,77.269,27.402,-157.6362,-25.1758,0.0000
C00648=51.954,75.301,26.968,-155.6180,-24.6145,0.0000
C00649=53.649,73.106,26.645,-153.4241,-23.6625,0.0000
C00650=56.833,70.280,26.515,-151.5463,-22.5146,0.0000
C00651=60.331,67.277,26.509,-151.7054,-22.8961,0.0000
C00652=63.901,63.901,26.513,-152.9991,-24.4188,0.0000
C00653=67.277,60.331,26.509,-154.3752,-25.8906,0.0000
C00654=70.280,56.833,26.515,-154.7574,-26.1118,0.0000
C00655=73.106,53.649,26.645,-153.8972,-24.1902,0.0000
C00656=75.301,51.954,26.968,-153.2978,-22.0434,0.0000
C00657=77.269,51.285,27.402,-153.0571,-20.1419,0.0000
C00658=79.281,51.105,27.838,-153.0681,-18.2227,0.0000
C00659=81.387,50.979,28.166,-153.3271,-15.9501,0.0000
C00660=83.570,50.396,28.327,-153.9815,-12.9075,0.0000
C00661=85.996,48.746,28.411,-155.8623,-9.2541,0.0000
C00662=88.332,46.201,28.479,-158.6259,-5.9076,0.0000
C00663=90.182,43.110,28.548,-161.3237,-3.6374,0.0000
C00664=91.693,39.893,28.594,-179.9961,-0.0088,0.0000
C00665=93.045,36.628,28.594,-179.9965,-0.0090,0.0000
C00666=94.252,33.285,28.548,169.1554,-15.7139,0.0000
C00667=95.129,29.791,28.479,168.7908,-19.2153,0.0000
C00668=95.277,26.340,28.411,169.2082,-23.5223,0.0000
C00669=94.728,23.458,28.327,170.6395,-27.4061,0.0000
C00670=93.597,21.502,28.166,172.6459,-29.9676,0.0000
C00671=92.196,19.923,27.838,174.3959,-31.6904,0.0000
C00672=90.901,18.373,27.402,176.0825,-32.9760,0.0000
C00673=89.983,16.509,26.968,177.9848,-34.0488,0.0000
C00674=89.629,13.759,26.645,-179.5835,-34.9980,0.0000
C00675=89.882,9.508,26.515,-177.1483,-35.5903,0.0000
C00676=90.233,4.912,26.509,-177.6240,-35.7234,0.0000
C00677=90.369,0.000,26.513,179.9995,-35.7771,0.0000
C00678=90.233,-4.912,26.509,177.6246,-35.7234,0.0000
C00679=89.882,-9.508,26.515,177.1492,-35.5903,0.0000
C00680=89.629,-13.759,26.645,179.5836,-34.9979,0.0000
C00681=89.983,-16.509,26.968,-177.9852,-34.0487,0.0000
C00682=90.901,-18.373,27.402,-176.0829,-32.9760,0.0000
C00683=92.196,-19.923,27.838,-174.3962,-31.6904,0.0000
C00684=93.597,-21.502,28.166,-172.6462,-29.9676,0.0000
C00685=94.728,-23.458,28.327,-170.6395,-27.4061,0.0000
C00686=95.277,-26.340,28.411,-169.2082,-23.5223,0.0000
C00687=95.129,-29.791,28.479,-168.7908,-19.2153,0.0000
C00688=94.252,-33.285,28.548,-169.1554,-15.7139,0.0000
C00689=93.045,-36.628,28.594,179.9965,-0.0090,0.0000
C00690=91.693,-39.893,28.594,179.9961,-0.0088,0.0000
C00691=90.182,-43.110,28.548,161.3237,-3.6374,0.0000
C00692=88.332,-46.201,28.479,158.6259,-5.9076,0.0000
C00693=85.996,-48.746,28.411,155.8623,-9.2541,0.0000
C00694=83.570,-50.396,28.327,153.9815,-12.9075,0.0000
C00695=81.387,-50.979,28.166,153.3270,-15.9500,0.0000
C00696=79.281,-51.105,27.838,153.0679,-18.2224,0.0000
C00697=77.269,-51.285,27.402,153.0568,-20.1417,0.0000
C00698=75.301,-51.954,26.968,153.2975,-22.0433,0.0000
C00699=73.106,-53.649,26.645,153.8971,-24.1904,0.0000
C00700=70.280,-56.833,26.515,154.7579,-26.1124,0.0000
C00701=67.277,-60.331,26.509,154.3756,-25.8909,0.0000
C00702=63.901,-63.901,26.513,152.9985,-24.4182,0.0000
C00703=60.331,-67.277,26.509,151.7057,-22.8965,0.0000
C00704=56.833,-70.280,26.515,151.5469,-22.5151,0.0000
C00705=53.649,-73.106,26.645,153.4242,-23.6625,0.0000
C00706=51.954,-75.301,26.968,155.6178,-24.6142,0.0000
C00707=51.285,-77.269,27.402,157.6360,-25.1755,0.0000
C00708=51.105,-79.281,27.838,159.7323,-25.4813,0.0000
C00709=50.979,-81.387,28.166,162.2637,-25.5701,0.0000
C00710=50.396,-83.570,28.327,165.6938,-25.3139,0.0000
C00711=48.746,-85.996,28.411,169.8768,-23.8040,0.0000
C00712=46.201,-88.332,28.479,173.6595,-21.2551,0.0000
C00713=43.110,-90.182,28.548,176.1610,-18.6373,0.0000
C00714=39.893,-91.693,28.594,179.9912,-0.0039,0.0000
C00715=36.628,-93.045,28.594,179.9910,-0.0035,0.0000
C00716=33.285,-94.252,28.548,164.0148,10.4347,0.0000
C00717=29.791,-95.129,28.479,160.4391,10.5773,0.0000
C00718=26.340,-95.277,28.411,156.1013,9.8857,0.0000
C00719=23.458,-94.728,28.327,152.2788,8.3021,0.0000
C00720=21.502,-93.597,28.166,149.8272,6.3665,0.0000
C00721=19.923,-92.196,27.838,148.1868,4.7664,0.0000
C00722=18.373,-90.901,27.402,146.9628,3.2856,0.0000
C00723=16.509,-89.983,26.968,145.9347,1.6696,0.0000
C00724=13.759,-89.629,26.645,145.0013,-0.3412,0.0000
C00725=9.508,-89.882,26.515,144.3761,-2.3187,0.0000
C00726=4.912,-90.233,26.509,144.2533,-1.9288,0.0000
C00727=0.000,-90.369,26.513,144.2229,0.0004,0.0000
C00728=0.000,-90.369,26.513,144.2229,0.0004,0.0000
C00729=-4.912,-90.233,26.509,144.2532,1.9283,0.0000
C00730=-9.508,-89.882,26.515,144.3761,2.3179,0.0000
C00731=-13.759,-89.629,26.645,145.0014,0.3411,0.0000
C00732=-16.509,-89.983,26.968,145.9348,-1.6693,0.0000
C00733=-18.373,-90.901,27.402,146.9628,-3.2853,0.0000
C00734=-19.923,-92.196,27.838,148.1868,-4.7661,0.0000
C00735=-21.502,-93.597,28.166,149.8272,-6.3663,0.0000
C00736=-23.458,-94.728,28.327,152.2788,-8.3020,0.0000
C00737=-26.340,-95.277,28.411,156.1013,-9.8857,0.0000
C00738=-29.791,-95.129,28.479,160.4391,-10.5773,0.0000
C00739=-33.285,-94.252,28.548,164.0148,-10.4347,0.0000
C00740=-36.628,-93.045,28.594,179.9910,0.0035,0.0000
C00741=-39.893,-91.693,28.594,179.9912,0.0039,0.0000
C00742=-43.110,-90.182,28.548,176.1610,18.6373,0.0000
C00743=-46.201,-88.332,28.479,173.6595,21.2551,0.0000
C00744=-48.746,-85.996,28.411,169.8768,23.8040,0.0000
C00745=-50.396,-83.570,28.327,165.6938,25.3139,0.0000
C00746=-50.979,-81.387,28.166,162.2638,25.5702,0.0000
C00747=-51.105,-79.281,27.838,159.7325,25.4815,0.0000
C00748=-51.285,-77.269,27.402,157.6362,25.1758,0.0000
C00749=-51.954,-75.301,26.968,155.6180,24.6145,0.0000
C00750=-53.649,-73.106,26.645,153.4241,23.6625,0.0000
C00751=-56.833,-70.280,26.515,151.5463,22.5146,0.0000
C00752=-60.331,-67.277,26.509,151.7054,22.8961,0.0000
C00753=-63.901,-63.901,26.513,152.9991,24.4188,0.0000
C00754=-67.277,-60.331,26.509,154.3752,25.8906,0.0000
C00755=-70.280,-56.833,26.515,154.7574,26.1118,0.0000
C00756=-73.106,-53.649,26.645,153.8972,24.1902,0.0000
C00757=-75.301,-51.954,26.968,153.2978,22.0434,0.0000
C00758=-77.269,-51.285,27.402,153.0571,20.1419,0.0000
C00759=-79.281,-51.105,27.838,153.0681,18.2227,0.0000
C00760=-81.387,-50.979,28.166,153.3271,15.9501,0.0000
C00761=-83.570,-50.396,28.327,153.9815,12.9075,0.0000
C00762=-85.996,-48.746,28.411,155.8623,9.2541,0.0000
C00763=-88.332,-46.201,28.479,158.6259,5.9076,0.0000
C00764=-90.182,-43.110,28.548,161.3237,3.6374,0.0000
C00765=-91.693,-39.893,28.594,179.9961,0.0088,0.0000
C00766=-93.045,-36.628,28.594,179.9965,0.0090,0.0000
C00767=-94.252,-33.285,28.548,-169.1554,15.7139,0.0000
C00768=-95.129,-29.791,28.479,-168.7908,19.2153,0.0000
C00769=-95.277,-26.340,28.411,-169.2082,23.5223,0.0000
C00770=-94.728,-23.458,28.327,-170.6395,27.4061,0.0000
C00771=-93.597,-21.502,28.166,-172.6459,29.9676,0.0000
C00772=-92.196,-19.923,27.838,-174.3959,31.6904,0.0000
C00773=-90.901,-18.373,27.402,-176.0825,32.9760,0.0000
C00774=-89.983,-16.509,26.968,-177.9848,34.0488,0.0000
C00775=-89.629,-13.759,26.645,179.5835,34.9980,0.0000
C00776=-89.882,-9.508,26.515,177.1483,35.5903,0.0000
C00777=-90.233,-4.912,26.509,177.6240,35.7234,0.0000
C00778=-90.369,0.000,26.513,-179.9995,35.7771,0.0000
C00779=-90.233,4.912,26.509,-177.6246,35.7234,0.0000
C00780=-89.882,9.508,26.515,-177.1492,35.5903,0.0000
C00781=-89.629,13.759,26.645,-179.5836,34.9979,0.0000
C00782=-89.983,16.509,26.968,177.9852,34.0487,0.0000
C00783=-90.901,18.373,27.402,176.0829,32.9760,0.0000
C00784=-92.196,19.923,27.838,174.3962,31.6904,0.0000
C00785=-93.597,21.502,28.166,172.6462,29.9676,0.0000
C00786=-94.728,23.458,28.327,170.6395,27.4061,0.0000
C00787=-95.277,26.340,28.411,169.2082,23.5223,0.0000
C00788=-95.129,29.791,28.479,168.7908,19.2153,0.0000
C00789=-94.252,33.285,28.548,169.1554,15.7139,0.0000
C00790=-93.045,36.628,28.594,-179.9965,0.0090,0.0000
C00791=-91.693,39.893,28.594,-179.9961,0.0088,0.0000
C00792=-90.182,43.110,28.548,-161.3237,3.6374,0.0000
C00793=-88.332,46.201,28.479,-158.6259,5.9076,0.0000
C00794=-85.996,48.746,28.411,-155.8623,9.2541,0.0000
C00795=-83.570,50.396,28.327,-153.9815,12.9075,0.0000
C00796=-81.387,50.979,28.166,-153.3270,15.9500,0.0000
C00797=-79.281,51.105,27.838,-153.0679,18.2224,0.0000
C00798=-77.269,51.285,27.402,-153.0568,20.1417,0.0000
C00799=-75.301,51.954,26.968,-153.2975,22.0433,0.0000
C00800=-73.106,53.649,26.645,-153.8971,24.1904,0.0000
C00801=-70.280,56.833,26.515,-154.7579,26.1124,0.0000
C00802=-67.277,60.331,26.509,-154.3756,25.8909,0.0000
C00803=-63.901,63.901,26.513,-152.9985,24.4182,0.0000
C00804=-60.331,67.277,26.509,-151.7057,22.8965,0.0000
C00805=-56.833,70.280,26.515,-151.5469,22.5151,0.0000
C00806=-53.649,73.106,26.645,-153.4242,23.6625,0.0000
C00807=-51.954,75.301,26.968,-155.6178,24.6142,0.0000
C00808=-51.285,77.269,27.402,-157.6360,25.1755,0.0000
C00809=-51.105,79.281,27.838,-159.7323,25.4813,0.0000
C00810=-50.979,81.387,28.166,-162.2637,25.5701,0.0000
C00811=-50.396,83.570,28.327,-165.6938,25.3139,0.0000
C00812=-48.746,85.996,28.411,-169.8768,23.8040,0.0000
C00813=-46.201,88.332,28.479,-173.6595,21.2551,0.0000
C00814=-43.110,90.182,28.548,-176.1610,18.6373,0.0000
C00815=-39.893,91.693,28.594,-179.9912,0.0039,0.0000
C00816=-36.628,93.045,28.594,-179.9910,0.0035,0.0000
C00817=-33.285,94.252,28.548,-164.0148,-10.4347,0.0000
C00818=-29.791,95.129,28.479,-160.4391,-10.5773,0.0000
C00819=-26.340,95.277,28.411,-156.1013,-9.8857,0.0000
C00820=-23.458,94.728,28.327,-152.2788,-8.3020,0.0000
C00821=-21.502,93.597,28.166,-149.8272,-6.3663,0.0000
C00822=-19.923,92.196,27.838,-148.1868,-4.7661,0.0000
C00823=-18.373,90.901,27.402,-146.9628,-3.2853,0.0000
C00824=-16.509,89.983,26.968,-145.9348,-1.6693,0.0000
C00825=-13.759,89.629,26.645,-145.0014,0.3411,0.0000
C00826=-9.508,89.882,26.515,-144.3761,2.3179,0.0000
C00827=-4.912,90.233,26.509,-144.2532,1.9283,0.0000
C00828=0.000,90.369,26.513,-144.2229,0.0004,0.0000
C00829=0.000,89.153,28.346,-143.5495,0.0004,0.0000
C00830=4.801,89.020,28.341,-143.5802,-1.9526,0.0000
C00831=9.321,88.681,28.348,-143.7013,-2.2454,0.0000
C00832=13.530,88.468,28.499,-144.3332,-0.0767,0.0000
C00833=16.227,88.922,28.874,-145.2729,2.0193,0.0000
C00834=18.049,89.999,29.382,-146.3100,3.6842,0.0000
C00835=19.567,91.502,29.895,-147.5648,5.2228,0.0000
C00836=21.117,93.139,30.283,-149.2771,6.8947,0.0000
C00837=23.038,94.499,30.474,-151.8791,8.9142,0.0000
C00838=25.943,95.229,30.574,-156.0777,10.7226,0.0000
C00839=29.476,95.186,30.656,-160.7880,11.3352,0.0000
C00840=33.085,94.318,30.738,-164.5494,11.0342,0.0000
C00841=36.560,93.071,30.793,-167.2361,10.3681,0.0000
C00842=39.959,91.663,30.793,-178.4228,-16.3158,0.0000
C00843=43.298,90.088,30.738,-177.0012,-18.6770,0.0000
C00844=46.464,88.150,30.656,-174.4993,-21.5385,0.0000
C00845=48.993,85.682,30.574,-170.5083,-24.4113,0.0000
C00846=50.531,83.111,30.474,-165.8486,-26.0291,0.0000
C00847=50.927,80.791,30.283,-162.2153,-26.3289,0.0000
C00848=50.865,78.538,29.895,-159.5560,-26.2345,0.0000
C00849=50.876,76.401,29.382,-157.3793,-25.9035,0.0000
C00850=51.403,74.351,28.874,-155.3078,-25.3079,0.0000
C00851=52.989,72.123,28.499,-153.0398,-24.2894,0.0000
C00852=56.115,69.298,28.348,-151.0224,-22.9904,0.0000
C00853=59.552,66.342,28.341,-151.1163,-23.2953,0.0000
C00854=63.040,63.040,28.346,-152.4228,-24.8420,0.0000
C00855=66.342,59.552,28.341,-153.8142,-26.3370,0.0000
C00856=69.298,56.115,28.348,-154.1264,-26.4858,0.0000
C00857=72.123,52.989,28.499,-153.1459,-24.4083,0.0000
C00858=74.351,51.403,28.874,-152.5053,-22.1884,0.0000
C00859=76.401,50.876,29.382,-152.2503,-20.2422,0.0000
C00860=78.538,50.865,29.895,-152.2588,-18.2592,0.0000
C00861=80.791,50.927,30.283,-152.5395,-15.8880,0.0000
C00862=83.111,50.531,30.474,-153.2681,-12.6907,0.0000
C00863=85.682,48.993,30.574,-155.2901,-8.6364,0.0000
C00864=88.150,46.464,30.656,-158.3711,-5.1156,0.0000
C00865=90.088,43.298,30.738,-161.2992,-2.8407,0.0000
C00866=91.663,39.959,30.793,-163.6783,-1.5136,0.0000
C00867=93.071,36.560,30.793,169.3751,-12.5521,0.0000
C00868=94.318,33.085,30.738,168.5628,-15.1580,0.0000
C00869=95.186,29.476,30.656,168.0151,-18.8230,0.0000
C00870=95.229,25.943,30.574,168.2963,-23.4793,0.0000
C00871=94.499,23.038,30.474,169.9157,-27.7517,0.0000
C00872=93.139,21.117,30.283,171.9932,-30.4770,0.0000
C00873=91.502,19.567,29.895,173.8188,-32.2842,0.0000
C00874=89.999,18.049,29.382,175.5749,-33.6111,0.0000
C00875=88.922,16.227,28.874,177.5435,-34.7025,0.0000
C00876=88.468,13.530,28.499,-179.9056,-35.6667,0.0000
C00877=88.681,9.321,28.348,-177.2147,-36.2664,0.0000
C00878=89.020,4.801,28.341,-177.5740,-36.3953,0.0000
C00879=89.153,0.000,28.346,179.9995,-36.4505,0.0000
C00880=89.020,-4.801,28.341,177.5746,-36.3953,0.0000
C00881=88.681,-9.321,28.348,177.2156,-36.2663,0.0000
C00882=88.468,-13.530,28.499,179.9057,-35.6666,0.0000
C00883=88.922,-16.227,28.874,-177.5438,-34.7024,0.0000
C00884=89.999,-18.049,29.382,-175.5753,-33.6111,0.0000
C00885=91.502,-19.567,29.895,-173.8192,-32.2842,0.0000
C00886=93.139,-21.117,30.283,-171.9935,-30.4771,0.0000
C00887=94.499,-23.038,30.474,-169.9158,-27.7517,0.0000
C00888=95.229,-25.943,30.574,-168.2963,-23.4793,0.0000
C00889=95.186,-29.476,30.656,-168.0151,-18.8230,0.0000
C00890=94.318,-33.085,30.738,-168.5628,-15.1580,0.0000
C00891=93.071,-36.560,30.793,-169.3751,-12.5521,0.0000
C00892=91.663,-39.959,30.793,163.6783,-1.5136,0.0000
C00893=90.088,-43.298,30.738,161.2992,-2.8407,0.0000
C00894=88.150,-46.464,30.656,158.3711,-5.1156,0.0000
C00895=85.682,-48.993,30.574,155.2901,-8.6364,0.0000
C00896=83.111,-50.531,30.474,153.2681,-12.6907,0.0000
C00897=80.791,-50.927,30.283,152.5393,-15.8878,0.0000
C00898=78.538,-50.865,29.895,152.2585,-18.2590,0.0000
C00899=76.401,-50.876,29.382,152.2501,-20.2419,0.0000
C00900=74.351,-51.403,28.874,152.5051,-22.1882,0.0000
C00901=72.123,-52.989,28.499,153.1460,-24.4085,0.0000
C00902=69.298,-56.115,28.348,154.1269,-26.4865,0.0000
C00903=66.342,-59.552,28.341,153.8146,-26.3374,0.0000
C00904=63.040,-63.040,28.346,152.4222,-24.8413,0.0000
C00905=59.552,-66.342,28.341,151.1166,-23.2958,0.0000
C00906=56.115,-69.298,28.348,151.0230,-22.9910,0.0000
C00907=52.989,-72.123,28.499,153.0399,-24.2894,0.0000
C00908=51.403,-74.351,28.874,155.3076,-25.3077,0.0000
C00909=50.876,-76.401,29.382,157.3791,-25.9032,0.0000
C00910=50.865,-78.538,29.895,159.5557,-26.2342,0.0000
C00911=50.927,-80.791,30.283,162.2151,-26.3288,0.0000
C00912=50.531,-83.111,30.474,165.8485,-26.0291,0.0000
C00913=48.993,-85.682,30.574,170.5083,-24.4113,0.0000
C00914=46.464,-88.150,30.656,174.4993,-21.5385,0.0000
C00915=43.298,-90.088,30.738,177.0012,-18.6770,0.0000
C00916=39.959,-91.663,30.793,178.4228,-16.3158,0.0000
C00917=36.560,-93.071,30.793,167.2361,10.3681,0.0000
C00918=33.085,-94.318,30.738,164.5494,11.0342,0.0000
C00919=29.476,-95.186,30.656,160.7880,11.3352,0.0000
C00920=25.943,-95.229,30.574,156.0777,10.7226,0.0000
C00921=23.038,-94.499,30.474,151.8791,8.9142,0.0000
C00922=21.117,-93.139,30.283,149.2771,6.8947,0.0000
C00923=19.567,-91.502,29.895,147.5648,5.2228,0.0000
C00924=18.049,-89.999,29.382,146.3100,3.6842,0.0000
C00925=16.227,-88.922,28.874,145.2729,2.0193,0.0000
C00926=13.530,-88.468,28.499,144.3332,-0.0767,0.0000
C00927=9.321,-88.681,28.348,143.7013,-2.2454,0.0000
C00928=4.801,-89.020,28.341,143.5802,-1.9526,0.0000
C00929=0.000,-89.153,28.346,143.5495,0.0004,0.0000
C00930=0.000,-89.153,28.346,143.5495,0.0004,0.0000
C00931=-4.801,-89.020,28.341,143.5801,1.9521,0.0000
C00932=-9.321,-88.681,28.348,143.7014,2.2447,0.0000
C00933=-13.530,-88.468,28.499,144.3333,0.0766,0.0000
C00934=-16.227,-88.922,28.874,145.2729,-2.0191,0.0000
C00935=-18.049,-89.999,29.382,146.3100,-3.6838,0.0000
C00936=-19.567,-91.502,29.895,147.5648,-5.2224,0.0000
C00937=-21.117,-93.139,30.283,149.2770,-6.8945,0.0000
C00938=-23.038,-94.499,30.474,151.8791,-8.9142,0.0000
C00939=-25.943,-95.229,30.574,156.0777,-10.7226,0.0000
C00940=-29.476,-95.186,30.656,160.7880,-11.3352,0.0000
C00941=-33.085,-94.318,30.738,164.5494,-11.0342,0.0000
C00942=-36.560,-93.071,30.793,167.2361,-10.3681,0.0000
C00943=-39.959,-91.663,30.793,178.4228,16.3158,0.0000
C00944=-43.298,-90.088,30.738,177.0012,18.6770,0.0000
C00945=-46.464,-88.150,30.656,174.4993,21.5385,0.0000
C00946=-48.993,-85.682,30.574,170.5083,24.4113,0.0000
C00947=-50.531,-83.111,30.474,165.8486,26.0291,0.0000
C00948=-50.927,-80.791,30.283,162.2153,26.3289,0.0000
C00949=-50.865,-78.538,29.895,159.5560,26.2345,0.0000
C00950=-50.876,-76.401,29.382,157.3793,25.9035,0.0000
C00951=-51.403,-74.351,28.874,155.3078,25.3079,0.0000
C00952=-52.989,-72.123,28.499,153.0398,24.2894,0.0000
C00953=-56.115,-69.298,28.348,151.0224,22.9904,0.0000
C00954=-59.552,-66.342,28.341,151.1163,23.2953,0.0000
C00955=-63.040,-63.040,28.346,152.4228,24.8420,0.0000
C00956=-66.342,-59.552,28.341,153.8142,26.3370,0.0000
C00957=-69.298,-56.115,28.348,154.1264,26.4858,0.0000
C00958=-72.123,-52.989,28.499,153.1459,24.4083,0.0000
C00959=-74.351,-51.403,28.874,152.5053,22.1884,0.0000
C00960=-76.401,-50.876,29.382,152.2503,20.2422,0.0000
C00961=-78.538,-50.865,29.895,152.2588,18.2592,0.0000
C00962=-80.791,-50.927,30.283,152.5395,15.8880,0.0000
C00963=-83.111,-50.531,30.474,153.2681,12.6907,0.0000
C00964=-85.682,-48.993,30.574,155.2901,8.6364,0.0000
C00965=-88.150,-46.464,30.656,158.3711,5.1156,0.0000
C00966=-90.088,-43.298,30.738,161.2992,2.8407,0.0000
C00967=-91.663,-39.959,30.793,163.6783,1.5136,0.0000
C00968=-93.071,-36.560,30.793,-169.3751,12.5521,0.0000
C00969=-94.318,-33.085,30.738,-168.5628,15.1580,0.0000
C00970=-95.186,-29.476,30.656,-168.0151,18.8230,0.0000
C00971=-95.229,-25.943,30.574,-168.2963,23.4793,0.0000
C00972=-94.499,-23.038,30.474,-169.9157,27.7517,0.0000
C00973=-93.139,-21.117,30.283,-171.9932,30.4770,0.0000
C00974=-91.502,-19.567,29.895,-173.8188,32.2842,0.0000
C00975=-89.999,-18.049,29.382,-175.5749,33.6111,0.0000
C00976=-88.922,-16.227,28.874,-177.5435,34.7025,0.0000
C00977=-88.468,-13.530,28.499,179.9056,35.6667,0.0000
C00978=-88.681,-9.321,28.348,177.2147,36.2664,0.0000
C00979=-89.020,-4.801,28.341,177.5740,36.3953,0.0000
C00980=-89.153,0.000,28.346,-179.9995,36.4505,0.0000
C00981=-89.020,4.801,28.341,-177.5746,36.3953,0.0000
C00982=-88.681,9.321,28.348,-177.2156,36.2663,0.0000
C00983=-88.468,13.530,28.499,-179.9057,35.6666,0.0000
C00984=-88.922,16.227,28.874,177.5438,34.7024,0.0000
C00985=-89.999,18.049,29.382,175.5753,33.6111,0.0000
C00986=-91.502,19.567,29.895,173.8192,32.2842,0.0000
C00987=-93.139,21.117,30.283,171.9935,30.4771,0.0000
C00988=-94.499,23.038,30.474,169.9158,27.7517,0.0000
C00989=-95.229,25.943,30.574,168.2963,23.4793,0.0000
C00990=-95.186,29.476,30.656,168.0151,18.8230,0.0000
C00991=-94.318,33.085,30.738,168.5628,15.1580,0.0000
C00992=-93.071,36.560,30.793,169.3751,12.5521,0.0000
C00993=-91.663,39.959,30.793,-163.6783,1.5136,0.0000
C00994=-90.088,43.298,30.738,-161.2992,2.8407,0.0000
C00995=-88.150,46.464,30.656,-158.3711,5.1156,0.0000
C00996=-85.682,48.993,30.574,-155.2901,8.6364,0.0000
C00997=-83.111,50.531,30.474,-153.2681,12.6907,0.0000
C00998=-80.791,50.927,30.283,-152.5393,15.8878,0.0000
C00999=-78.538,50.865,29.895,-152.2585,18.2590,0.0000
C01000=-76.401,50.876,29.382,-152.2501,20.2419,0.0000
C01001=-74.351,51.403,28.874,-152.5051,22.1882,0.0000
C01002=-72.123,52.989,28.499,-153.1460,24.4085,0.0000
C01003=-69.298,56.115,28.348,-154.1269,26.4865,0.0000
C01004=-66.342,59.552,28.341,-153.8146,26.3374,0.0000
C01005=-63.040,63.040,28.346,-152.4222,24.8413,0.0000
C01006=-59.552,66.342,28.341,-151.1166,23.2958,0.0000
C01007=-56.115,69.298,28.348,-151.0230,22.9910,0.0000
C01008=-52.989,72.123,28.499,-153.0399,24.2894,0.0000
C01009=-51.403,74.351,28.874,-155.3076,25.3077,0.0000
C01010=-50.876,76.401,29.382,-157.3791,25.9032,0.0000
C01011=-50.865,78.538,29.895,-159.5557,26.2342,0.0000
C01012=-50.927,80.791,30.283,-162.2151,26.3288,0.0000
C01013=-50.531,83.111,30.474,-165.8485,26.0291,0.0000
C01014=-48.993,85.682,30.574,-170.5083,24.4113,0.0000
C01015=-46.464,88.150,30.656,-174.4993,21.5385,0.0000
C01016=-43.298,90.088,30.738,-177.0012,18.6770,0.0000
C01017=-39.959,91.663,30.793,-178.4228,16.3158,0.0000
C01018=-36.560,93.071,30.793,-167.2361,-10.3681,0.0000
C01019=-33.085,94.318,30.738,-164.5494,-11.0342,0.0000
C01020=-29.476,95.186,30.656,-160.7880,-11.3352,0.0000
C01021=-25.943,95.229,30.574,-156.0777,-10.7226,0.0000
C01022=-23.038,94.499,30.474,-151.8791,-8.9142,0.0000
C01023=-21.117,93.139,30.283,-149.2770,-6.8945,0.0000
C01024=-19.567,91.502,29.895,-147.5648,-5.2224,0.0000
C01025=-18.049,89.999,29.382,-146.3100,-3.6838,0.0000
C01026=-16.227,88.922,28.874,-145.2729,-2.0191,0.0000
C01027=-13.530,88.468,28.499,-144.3333,0.0766,0.0000
C01028=-9.321,88.681,28.348,-143.7014,2.2447,0.0000
C01029=-4.801,89.020,28.341,-143.5801,1.9521,0.0000
C01030=0.000,89.153,28.346,-143.5495,0.0004,0.0000
C01031=0.000,87.904,30.157,-142.9665,0.0004,0.0000
C01032=4.687,87.776,30.152,-142.9974,-1.9709,0.0000
C01033=9.129,87.447,30.160,-143.1172,-2.1665,0.0000
C01034=13.294,87.274,30.332,-143.7584,0.1810,0.0000
C01035=15.938,87.830,30.762,-144.7049,2.3495,0.0000
C01036=17.714,89.068,31.347,-145.7504,4.0563,0.0000
C01037=19.200,90.783,31.942,-147.0359,5.6502,0.0000
C01038=20.718,92.664,32.394,-148.8239,7.3963,0.0000
C01039=22.602,94.262,32.617,-151.5923,9.5064,0.0000
C01040=25.531,95.180,32.735,-156.2418,11.5105,0.0000
C01041=29.149,95.246,32.831,-161.3668,11.9813,0.0000
C01042=32.878,94.386,32.928,-165.3054,11.4655,0.0000
C01043=36.490,93.098,32.991,-167.9997,10.6450,0.0000
C01044=40.028,91.633,32.991,-179.1734,-15.9684,0.0000
C01045=43.493,89.989,32.928,-177.8716,-18.4421,0.0000
C01046=46.737,87.960,32.831,-175.4225,-21.5797,0.0000
C01047=49.249,85.356,32.735,-171.2494,-24.8504,0.0000
C01048=50.671,82.635,32.617,-166.0806,-26.6517,0.0000
C01049=50.874,80.174,32.394,-162.2267,-27.0025,0.0000
C01050=50.617,77.770,31.942,-159.4344,-26.9039,0.0000
C01051=50.455,75.506,31.347,-157.1795,-26.5501,0.0000
C01052=50.836,73.375,30.762,-155.0605,-25.9255,0.0000
C01053=52.312,71.113,30.332,-152.7270,-24.8515,0.0000
C01054=55.379,68.290,30.160,-150.5760,-23.4130,0.0000
C01055=58.753,65.381,30.152,-150.6047,-23.6409,0.0000
C01056=62.157,62.157,30.157,-151.9207,-25.2066,0.0000
C01057=65.381,58.753,30.152,-153.3236,-26.7203,0.0000
C01058=68.290,55.379,30.160,-153.5659,-26.7956,0.0000
C01059=71.113,52.312,30.332,-152.4767,-24.5694,0.0000
C01060=73.375,50.836,30.762,-151.8038,-22.2859,0.0000
C01061=75.506,50.455,31.347,-151.5378,-20.3008,0.0000
C01062=77.770,50.617,31.942,-151.5446,-18.2561,0.0000
C01063=80.174,50.874,32.394,-151.8479,-15.7821,0.0000
C01064=82.635,50.671,32.617,-152.6577,-12.4155,0.0000
C01065=85.356,49.249,32.735,-154.8928,-7.9348,0.0000
C01066=87.960,46.737,32.831,-158.3577,-4.2561,0.0000
C01067=89.989,43.493,32.928,-161.5460,-2.0191,0.0000
C01068=91.633,40.028,32.991,-164.0300,-0.7947,0.0000
C01069=93.098,36.490,32.991,169.1228,-11.7907,0.0000
C01070=94.386,32.878,32.928,168.1576,-14.3949,0.0000
C01071=95.246,29.149,32.831,167.3767,-18.2128,0.0000
C01072=95.180,25.531,32.735,167.4561,-23.2520,0.0000
C01073=94.262,22.602,32.617,169.2209,-27.9830,0.0000
C01074=92.664,20.718,32.394,171.3727,-30.8881,0.0000
C01075=90.783,19.200,31.942,173.2748,-32.7838,0.0000
C01076=89.068,17.714,31.347,175.0965,-34.1520,0.0000
C01077=87.830,15.938,30.762,177.1222,-35.2610,0.0000
C01078=87.274,13.294,30.332,179.7756,-36.2414,0.0000
C01079=87.447,9.129,30.160,-177.2921,-36.8521,0.0000
C01080=87.776,4.687,30.152,-177.5326,-36.9771,0.0000
C01081=87.904,0.000,30.157,179.9995,-37.0335,0.0000
C01082=87.776,-4.687,30.152,177.5332,-36.9771,0.0000
C01083=87.447,-9.130,30.160,177.2931,-36.8520,0.0000
C01084=87.274,-13.294,30.332,-179.7753,-36.2413,0.0000
C01085=87.830,-15.938,30.762,-177.1225,-35.2609,0.0000
C01086=89.068,-17.714,31.347,-175.0970,-34.1520,0.0000
C01087=90.783,-19.200,31.942,-173.2752,-32.7838,0.0000
C01088=92.664,-20.718,32.394,-171.3730,-30.8882,0.0000
C01089=94.262,-22.602,32.617,-169.2210,-27.9830,0.0000
C01090=95.180,-25.531,32.735,-167.4561,-23.2520,0.0000
C01091=95.246,-29.149,32.831,-167.3767,-18.2128,0.0000
C01092=94.386,-32.878,32.928,-168.1576,-14.3949,0.0000
C01093=93.098,-36.490,32.991,-169.1228,-11.7907,0.0000
C01094=91.633,-40.028,32.991,164.0300,-0.7947,0.0000
C01095=89.989,-43.493,32.928,161.5460,-2.0191,0.0000
C01096=87.960,-46.737,32.831,158.3577,-4.2561,0.0000
C01097=85.356,-49.249,32.735,154.8928,-7.9348,0.0000
C01098=82.635,-50.671,32.617,152.6577,-12.4154,0.0000
C01099=80.174,-50.874,32.394,151.8478,-15.7819,0.0000
C01100=77.770,-50.617,31.942,151.5444,-18.2558,0.0000
C01101=75.506,-50.455,31.347,151.5375,-20.3005,0.0000
C01102=73.375,-50.836,30.762,151.8036,-22.2858,0.0000
C01103=71.113,-52.312,30.332,152.4768,-24.5697,0.0000
C01104=68.290,-55.379,30.160,153.5664,-26.7963,0.0000
C01105=65.381,-58.753,30.152,153.3239,-26.7206,0.0000
C01106=62.157,-62.157,30.157,151.9201,-25.2059,0.0000
C01107=58.753,-65.381,30.152,150.6050,-23.6413,0.0000
C01108=55.379,-68.290,30.160,150.5766,-23.4136,0.0000
C01109=52.312,-71.113,30.332,152.7272,-24.8515,0.0000
C01110=50.836,-73.375,30.762,155.0604,-25.9252,0.0000
C01111=50.455,-75.506,31.347,157.1793,-26.5499,0.0000
C01112=50.617,-77.770,31.942,159.4341,-26.9036,0.0000
C01113=50.874,-80.174,32.394,162.2264,-27.0024,0.0000
C01114=50.671,-82.635,32.617,166.0805,-26.6516,0.0000
C01115=49.249,-85.356,32.735,171.2494,-24.8504,0.0000
C01116=46.737,-87.960,32.831,175.4225,-21.5797,0.0000
C01117=43.493,-89.989,32.928,177.8716,-18.4421,0.0000
C01118=40.028,-91.633,32.991,179.1734,-15.9684,0.0000
C01119=36.490,-93.098,32.991,167.9997,10.6450,0.0000
C01120=32.878,-94.386,32.928,165.3054,11.4655,0.0000
C01121=29.149,-95.246,32.831,161.3668,11.9813,0.0000
C01122=25.531,-95.180,32.735,156.2418,11.5105,0.0000
C01123=22.602,-94.262,32.617,151.5923,9.5064,0.0000
C01124=20.718,-92.664,32.394,148.8239,7.3963,0.0000
C01125=19.200,-90.783,31.942,147.0359,5.6502,0.0000
C01126=17.714,-89.068,31.347,145.7504,4.0563,0.0000
C01127=15.938,-87.830,30.762,144.7049,2.3495,0.0000
C01128=13.294,-87.274,30.332,143.7584,0.1810,0.0000
C01129=9.129,-87.447,30.160,143.1172,-2.1665,0.0000
C01130=4.687,-87.776,30.152,142.9974,-1.9709,0.0000
C01131=0.000,-87.904,30.157,142.9665,0.0004,0.0000
C01132=0.000,-87.904,30.157,142.9665,0.0004,0.0000
C01133=-4.687,-87.776,30.152,142.9973,1.9704,0.0000
C01134=-9.130,-87.447,30.160,143.1173,2.1657,0.0000
C01135=-13.294,-87.274,30.332,143.7585,-0.1812,0.0000
C01136=-15.938,-87.830,30.762,144.7050,-2.3492,0.0000
C01137=-17.714,-89.068,31.347,145.7504,-4.0559,0.0000
C01138=-19.200,-90.783,31.942,147.0359,-5.6498,0.0000
C01139=-20.718,-92.664,32.394,148.8238,-7.3960,0.0000
C01140=-22.602,-94.262,32.617,151.5922,-9.5063,0.0000
C01141=-25.531,-95.180,32.735,156.2418,-11.5105,0.0000
C01142=-29.149,-95.246,32.831,161.3668,-11.9813,0.0000
C01143=-32.878,-94.386,32.928,165.3054,-11.4655,0.0000
C01144=-36.490,-93.098,32.991,167.9997,-10.6450,0.0000
C01145=-40.028,-91.633,32.991,179.1734,15.9684,0.0000
C01146=-43.493,-89.989,32.928,177.8716,18.4421,0.0000
C01147=-46.737,-87.960,32.831,175.4225,21.5797,0.0000
C01148=-49.249,-85.356,32.735,171.2494,24.8504,0.0000
C01149=-50.671,-82.635,32.617,166.0806,26.6517,0.0000
C01150=-50.874,-80.174,32.394,162.2267,27.0025,0.0000
C01151=-50.617,-77.770,31.942,159.4344,26.9039,0.0000
C01152=-50.455,-75.506,31.347,157.1795,26.5501,0.0000
C01153=-50.836,-73.375,30.762,155.0605,25.9255,0.0000
C01154=-52.312,-71.113,30.332,152.7270,24.8515,0.0000
C01155=-55.379,-68.290,30.160,150.5760,23.4130,0.0000
C01156=-58.753,-65.381,30.152,150.6047,23.6409,0.0000
C01157=-62.157,-62.157,30.157,151.9207,25.2066,0.0000
C01158=-65.381,-58.753,30.152,153.3236,26.7203,0.0000
C01159=-68.290,-55.379,30.160,153.5659,26.7956,0.0000
C01160=-71.113,-52.312,30.332,152.4767,24.5694,0.0000
C01161=-73.375,-50.836,30.762,151.8038,22.2859,0.0000
C01162=-75.506,-50.455,31.347,151.5378,20.3008,0.0000
C01163=-77.770,-50.617,31.942,151.5446,18.2561,0.0000
C01164=-80.174,-50.874,32.394,151.8479,15.7821,0.0000
C01165=-82.635,-50.671,32.617,152.6577,12.4155,0.0000
C01166=-85.356,-49.249,32.735,154.8928,7.9348,0.0000
C01167=-87.960,-46.737,32.831,158.3577,4.2561,0.0000
C01168=-89.989,-43.493,32.928,161.5460,2.0191,0.0000
C01169=-91.633,-40.028,32.991,164.0300,0.7947,0.0000
C01170=-93.098,-36.490,32.991,-169.1228,11.7907,0.0000
C01171=-94.386,-32.878,32.928,-168.1576,14.3949,0.0000
C01172=-95.246,-29.149,32.831,-167.3767,18.2128,0.0000
C01173=-95.180,-25.531,32.735,-167.4561,23.2520,0.0000
C01174=-94.262,-22.602,32.617,-169.2209,27.9830,0.0000
C01175=-92.664,-20.718,32.394,-171.3727,30.8881,0.0000
C01176=-90.783,-19.200,31.942,-173.2748,32.7838,0.0000
C01177=-89.068,-17.714,31.347,-175.0965,34.1520,0.0000
C01178=-87.830,-15.938,30.762,-177.1222,35.2610,0.0000
C01179=-87.274,-13.294,30.332,-179.7756,36.2414,0.0000
C01180=-87.447,-9.129,30.160,177.2921,36.8521,0.0000
C01181=-87.776,-4.687,30.152,177.5326,36.9771,0.0000
C01182=-87.904,0.000,30.157,-179.9995,37.0335,0.0000
C01183=-87.776,4.687,30.152,-177.5332,36.9771,0.0000
C01184=-87.447,9.130,30.160,-177.2931,36.8520,0.0000
C01185=-87.274,13.294,30.332,179.7753,36.2413,0.0000
C01186=-87.830,15.938,30.762,177.1225,35.2609,0.0000
C01187=-89.068,17.714,31.347,175.0970,34.1520,0.0000
C01188=-90.783,19.200,31.942,173.2752,32.7838,0.0000
C01189=-92.664,20.718,32.394,171.3730,30.8882,0.0000
C01190=-94.262,22.602,32.617,169.2210,27.9830,0.0000
C01191=-95.180,25.531,32.735,167.4561,23.2520,0.0000
C01192=-95.246,29.149,32.831,167.3767,18.2128,0.0000
C01193=-94.386,32.878,32.928,168.1576,14.3949,0.0000
C01194=-93.098,36.490,32.991,169.1228,11.7907,0.0000
C01195=-91.633,40.028,32.991,-164.0300,0.7947,0.0000
C01196=-89.989,43.493,32.928,-161.5460,2.0191,0.0000
C01197=-87.960,46.737,32.831,-158.3577,4.2561,0.0000
C01198=-85.356,49.249,32.735,-154.8928,7.9348,0.0000
C01199=-82.635,50.671,32.617,-152.6577,12.4154,0.0000
C01200=-80.174,50.874,32.394,-151.8478,15.7819,0.0000
C01201=-77.770,50.617,31.942,-151.5444,18.2558,0.0000
C01202=-75.506,50.455,31.347,-151.5375,20.3005,0.0000
C01203=-73.375,50.836,30.762,-151.8036,22.2858,0.0000
C01204=-71.113,52.312,30.332,-152.4768,24.5697,0.0000
C01205=-68.290,55.379,30.160,-153.5664,26.7963,0.0000
C01206=-65.381,58.753,30.152,-153.3239,26.7206,0.0000
C01207=-62.157,62.157,30.157,-151.9201,25.2059,0.0000
C01208=-58.753,65.381,30.152,-150.6050,23.6413,0.0000
C01209=-55.379,68.290,30.160,-150.5766,23.4136,0.0000
C01210=-52.312,71.113,30.332,-152.7272,24.8515,0.0000
C01211=-50.836,73.375,30.762,-155.0604,25.9252,0.0000
C01212=-50.455,75.506,31.347,-157.1793,26.5499,0.0000
C01213=-50.617,77.770,31.942,-159.4341,26.9036,0.0000
C01214=-50.874,80.174,32.394,-162.2264,27.0024,0.0000
C01215=-50.671,82.635,32.617,-166.0805,26.6516,0.0000
C01216=-49.249,85.356,32.735,-171.2494,24.8504,0.0000
C01217=-46.737,87.960,32.831,-175.4225,21.5797,0.0000
C01218=-43.493,89.989,32.928,-177.8716,18.4421,0.0000
C01219=-40.028,91.633,32.991,-179.1734,15.9684,0.0000
C01220=-36.490,93.098,32.991,-167.9997,-10.6450,0.0000
C01221=-32.878,94.386,32.928,-165.3054,-11.4655,0.0000
C01222=-29.149,95.246,32.831,-161.3668,-11.9813,0.0000
C01223=-25.531,95.180,32.735,-156.2418,-11.5105,0.0000
C01224=-22.602,94.262,32.617,-151.5922,-9.5063,0.0000
C01225=-20.718,92.664,32.394,-148.8238,-7.3960,0.0000
C01226=-19.200,90.783,31.942,-147.0359,-5.6498,0.0000
C01227=-17.714,89.068,31.347,-145.7504,-4.0559,0.0000
C01228=-15.938,87.830,30.762,-144.7050,-2.3492,0.0000
C01229=-13.294,87.274,30.332,-143.7585,-0.1812,0.0000
C01230=-9.130,87.447,30.160,-143.1173,2.1657,0.0000
C01231=-4.687,87.776,30.152,-142.9973,1.9704,0.0000
C01232=0.000,87.904,30.157,-142.9665,0.0004,0.0000
C01233=0.000,86.627,31.948,-142.4647,0.0004,0.0000
C01234=4.570,86.503,31.943,-142.4958,-1.9843,0.0000
C01235=8.933,86.186,31.951,-142.6146,-2.0836,0.0000
C01236=13.053,86.053,32.146,-143.2671,0.4302,0.0000
C01237=15.641,86.712,32.633,-144.2202,2.6593,0.0000
C01238=17.370,88.113,33.299,-145.2726,4.4018,0.0000
C01239=18.822,90.045,33.980,-146.5883,6.0491,0.0000
C01240=20.308,92.176,34.500,-148.4570,7.8751,0.0000
C01241=22.152,94.017,34.757,-151.4108,10.0814,0.0000
C01242=25.107,95.129,34.893,-156.5929,12.2478,0.0000
C01243=28.812,95.307,35.004,-162.1672,12.5020,0.0000
C01244=32.664,94.457,35.116,-166.2550,11.7175,0.0000
C01245=36.417,93.126,35.190,-168.9188,10.7245,0.0000
C01246=40.099,91.601,35.190,-179.8842,-15.3738,0.0000
C01247=43.694,89.888,35.116,-178.7409,-17.9455,0.0000
C01248=47.019,87.765,35.004,-176.4080,-21.3756,0.0000
C01249=49.513,85.019,34.893,-172.0960,-25.1202,0.0000
C01250=50.816,82.144,34.757,-166.3863,-27.1886,0.0000
C01251=50.818,79.538,34.500,-162.2926,-27.6009,0.0000
C01252=50.362,76.980,33.980,-159.3591,-27.4979,0.0000
C01253=50.022,74.588,33.299,-157.0282,-27.1230,0.0000
C01254=50.255,72.374,32.633,-154.8679,-26.4737,0.0000
C01255=51.619,70.079,32.146,-152.4774,-25.3539,0.0000
C01256=54.626,67.259,31.951,-150.1996,-23.7874,0.0000
C01257=57.935,64.399,31.943,-150.1637,-23.9386,0.0000
C01258=61.254,61.254,31.948,-151.4862,-25.5189,0.0000
C01259=64.398,57.936,31.943,-152.8970,-27.0470,0.0000
C01260=67.259,54.626,31.951,-153.0707,-27.0489,0.0000
C01261=70.079,51.619,32.146,-151.8835,-24.6822,0.0000
C01262=72.374,50.255,32.633,-151.1856,-22.3445,0.0000
C01263=74.588,50.022,33.299,-150.9108,-20.3262,0.0000
C01264=76.980,50.362,33.980,-150.9163,-18.2215,0.0000
C01265=79.538,50.818,34.500,-151.2418,-15.6373,0.0000
C01266=82.144,50.816,34.757,-152.1423,-12.0854,0.0000
C01267=85.019,49.513,34.893,-154.6689,-7.1523,0.0000
C01268=87.765,47.019,35.004,-158.5862,-3.3446,0.0000
C01269=89.888,43.694,35.116,-162.0504,-1.1979,0.0000
C01270=91.601,40.099,35.190,-164.6262,-0.1116,0.0000
C01271=93.126,36.417,35.190,169.0766,-10.8852,0.0000
C01272=94.457,32.664,35.116,167.9470,-13.4532,0.0000
C01273=95.307,28.812,35.004,166.8884,-17.3963,0.0000
C01274=95.129,25.107,34.893,166.6914,-22.8438,0.0000
C01275=94.017,22.152,34.757,168.5535,-28.1081,0.0000
C01276=92.176,20.308,34.500,170.7813,-31.2119,0.0000
C01277=90.045,18.822,33.980,172.7650,-33.2015,0.0000
C01278=88.113,17.370,33.299,174.6492,-34.6103,0.0000
C01279=86.712,15.641,32.633,176.7232,-35.7353,0.0000
C01280=86.053,13.053,32.146,179.4632,-36.7317,0.0000
C01281=86.186,8.933,31.951,-177.3784,-37.3564,0.0000
C01282=86.503,4.570,31.943,-177.4993,-37.4778,0.0000
C01283=86.627,0.000,31.948,179.9995,-37.5353,0.0000
C01284=86.503,-4.570,31.943,177.4999,-37.4779,0.0000
C01285=86.186,-8.933,31.951,177.3795,-37.3564,0.0000
C01286=86.053,-13.053,32.146,-179.4629,-36.7316,0.0000
C01287=86.712,-15.641,32.633,-176.7235,-35.7353,0.0000
C01288=88.113,-17.370,33.299,-174.6496,-34.6103,0.0000
C01289=90.045,-18.822,33.980,-172.7654,-33.2016,0.0000
C01290=92.176,-20.308,34.500,-170.7817,-31.2120,0.0000
C01291=94.017,-22.152,34.757,-168.5537,-28.1082,0.0000
C01292=95.129,-25.107,34.893,-166.6914,-22.8438,0.0000
C01293=95.307,-28.812,35.004,-166.8884,-17.3963,0.0000
C01294=94.457,-32.664,35.116,-167.9470,-13.4532,0.0000
C01295=93.126,-36.417,35.190,-169.0766,-10.8852,0.0000
C01296=91.601,-40.099,35.190,164.6262,-0.1116,0.0000
C01297=89.888,-43.694,35.116,162.0504,-1.1979,0.0000
C01298=87.765,-47.019,35.004,158.5862,-3.3446,0.0000
C01299=85.019,-49.513,34.893,154.6689,-7.1523,0.0000
C01300=82.144,-50.816,34.757,152.1423,-12.0853,0.0000
C01301=79.538,-50.818,34.500,151.2416,-15.6370,0.0000
C01302=76.980,-50.362,33.980,150.9161,-18.2212,0.0000
C01303=74.588,-50.022,33.299,150.9105,-20.3259,0.0000
C01304=72.374,-50.255,32.633,151.1854,-22.3443,0.0000
C01305=70.079,-51.619,32.146,151.8836,-24.6825,0.0000
C01306=67.259,-54.626,31.951,153.0712,-27.0495,0.0000
C01307=64.399,-57.935,31.943,152.8974,-27.0473,0.0000
C01308=61.254,-61.254,31.948,151.4856,-25.5183,0.0000
C01309=57.936,-64.398,31.943,150.1640,-23.9390,0.0000
C01310=54.626,-67.259,31.951,150.2002,-23.7880,0.0000
C01311=51.619,-70.079,32.146,152.4777,-25.3540,0.0000
C01312=50.255,-72.374,32.633,154.8677,-26.4735,0.0000
C01313=50.022,-74.588,33.299,157.0279,-27.1227,0.0000
C01314=50.362,-76.980,33.980,159.3588,-27.4977,0.0000
C01315=50.818,-79.538,34.500,162.2923,-27.6007,0.0000
C01316=50.816,-82.144,34.757,166.3861,-27.1886,0.0000
C01317=49.513,-85.019,34.893,172.0960,-25.1202,0.0000
C01318=47.019,-87.765,35.004,176.4080,-21.3756,0.0000
C01319=43.694,-89.888,35.116,178.7409,-17.9455,0.0000
C01320=40.099,-91.601,35.190,179.8842,-15.3738,0.0000
C01321=36.417,-93.126,35.190,168.9188,10.7245,0.0000
C01322=32.664,-94.457,35.116,166.2550,11.7175,0.0000
C01323=28.812,-95.307,35.004,162.1672,12.5020,0.0000
C01324=25.107,-95.129,34.893,156.5929,12.2478,0.0000
C01325=22.152,-94.017,34.757,151.4108,10.0814,0.0000
C01326=20.308,-92.176,34.500,148.4570,7.8751,0.0000
C01327=18.822,-90.045,33.980,146.5883,6.0491,0.0000
C01328=17.370,-88.113,33.299,145.2726,4.4018,0.0000
C01329=15.641,-86.712,32.633,144.2202,2.6593,0.0000
C01330=13.053,-86.053,32.146,143.2671,0.4302,0.0000
C01331=8.933,-86.186,31.951,142.6146,-2.0836,0.0000
C01332=4.570,-86.503,31.943,142.4958,-1.9843,0.0000
C01333=0.000,-86.627,31.948,142.4647,0.0004,0.0000
C01334=0.000,-86.627,31.948,142.4647,0.0004,0.0000
C01335=-4.570,-86.503,31.943,142.4957,1.9838,0.0000
C01336=-8.933,-86.186,31.951,142.6147,2.0827,0.0000
C01337=-13.053,-86.053,32.146,143.2672,-0.4305,0.0000
C01338=-15.641,-86.712,32.633,144.2203,-2.6591,0.0000
C01339=-17.370,-88.113,33.299,145.2726,-4.4015,0.0000
C01340=-18.822,-90.045,33.980,146.5883,-6.0487,0.0000
C01341=-20.308,-92.176,34.500,148.4569,-7.8748,0.0000
C01342=-22.152,-94.017,34.757,151.4108,-10.0813,0.0000
C01343=-25.107,-95.129,34.893,156.5929,-12.2478,0.0000
C01344=-28.812,-95.307,35.004,162.1672,-12.5020,0.0000
C01345=-32.664,-94.457,35.116,166.2550,-11.7175,0.0000
C01346=-36.417,-93.126,35.190,168.9188,-10.7245,0.0000
C01347=-40.099,-91.601,35.190,179.8842,15.3738,0.0000
C01348=-43.694,-89.888,35.116,178.7409,17.9455,0.0000
C01349=-47.019,-87.765,35.004,176.4080,21.3756,0.0000
C01350=-49.513,-85.019,34.893,172.0960,25.1202,0.0000
C01351=-50.816,-82.144,34.757,166.3863,27.1886,0.0000
C01352=-50.818,-79.538,34.500,162.2926,27.6009,0.0000
C01353=-50.362,-76.980,33.980,159.3591,27.4979,0.0000
C01354=-50.022,-74.588,33.299,157.0282,27.1230,0.0000
C01355=-50.255,-72.374,32.633,154.8679,26.4737,0.0000
C01356=-51.619,-70.079,32.146,152.4774,25.3539,0.0000
C01357=-54.626,-67.259,31.951,150.1996,23.7874,0.0000
C01358=-57.935,-64.399,31.943,150.1637,23.9386,0.0000
C01359=-61.254,-61.254,31.948,151.4862,25.5189,0.0000
C01360=-64.398,-57.936,31.943,152.8970,27.0470,0.0000
C01361=-67.259,-54.626,31.951,153.0707,27.0489,0.0000
C01362=-70.079,-51.619,32.146,151.8835,24.6822,0.0000
C01363=-72.374,-50.255,32.633,151.1856,22.3445,0.0000
C01364=-74.588,-50.022,33.299,150.9108,20.3262,0.0000
C01365=-76.980,-50.362,33.980,150.9163,18.2215,0.0000
C01366=-79.538,-50.818,34.500,151.2418,15.6373,0.0000
C01367=-82.144,-50.816,34.757,152.1423,12.0854,0.0000
C01368=-85.019,-49.513,34.893,154.6689,7.1523,0.0000
C01369=-87.765,-47.019,35.004,158.5862,3.3446,0.0000
C01370=-89.888,-43.694,35.116,162.0504,1.1979,0.0000
C01371=-91.601,-40.099,35.190,164.6262,0.1116,0.0000
C01372=-93.126,-36.417,35.190,-169.0766,10.8852,0.0000
C01373=-94.457,-32.664,35.116,-167.9470,13.4532,0.0000
C01374=-95.307,-28.812,35.004,-166.8884,17.3963,0.0000
C01375=-95.129,-25.107,34.893,-166.6914,22.8438,0.0000
C01376=-94.017,-22.152,34.757,-168.5535,28.1081,0.0000
C01377=-92.176,-20.308,34.500,-170.7813,31.2119,0.0000
C01378=-90.045,-18.822,33.980,-172.7650,33.2015,0.0000
C01379=-88.113,-17.370,33.299,-174.6492,34.6103,0.0000
C01380=-86.712,-15.641,32.633,-176.7232,35.7353,0.0000
C01381=-86.053,-13.053,32.146,-179.4632,36.7317,0.0000
C01382=-86.186,-8.933,31.951,177.3784,37.3564,0.0000
C01383=-86.503,-4.570,31.943,177.4993,37.4778,0.0000
C01384=-86.627,0.000,31.948,-179.9995,37.5353,0.0000
C01385=-86.503,4.570,31.943,-177.4999,37.4779,0.0000
C01386=-86.186,8.933,31.951,-177.3795,37.3564,0.0000
C01387=-86.053,13.053,32.146,179.4629,36.7316,0.0000
C01388=-86.712,15.641,32.633,176.7235,35.7353,0.0000
C01389=-88.113,17.370,33.299,174.6496,34.6103,0.0000
C01390=-90.045,18.822,33.980,172.7654,33.2016,0.0000
C01391=-92.176,20.308,34.500,170.7817,31.2120,0.0000
C01392=-94.017,22.152,34.757,168.5537,28.1082,0.0000
C01393=-95.129,25.107,34.893,166.6914,22.8438,0.0000
C01394=-95.307,28.812,35.004,166.8884,17.3963,0.0000
C01395=-94.457,32.664,35.116,167.9470,13.4532,0.0000
C01396=-93.126,36.417,35.190,169.0766,10.8852,0.0000
C01397=-91.601,40.099,35.190,-164.6262,0.1116,0.0000
C01398=-89.888,43.694,35.116,-162.0504,1.1979,0.0000
C01399=-87.765,47.019,35.004,-158.5862,3.3446,0.0000
C01400=-85.019,49.513,34.893,-154.6689,7.1523,0.0000
C01401=-82.144,50.816,34.757,-152.1423,12.0853,0.0000
C01402=-79.538,50.818,34.500,-151.2416,15.6370,0.0000
C01403=-76.980,50.362,33.980,-150.9161,18.2212,0.0000
C01404=-74.588,50.022,33.299,-150.9105,20.3259,0.0000
C01405=-72.374,50.255,32.633,-151.1854,22.3443,0.0000
C01406=-70.079,51.619,32.146,-151.8836,24.6825,0.0000
C01407=-67.259,54.626,31.951,-153.0712,27.0495,0.0000
C01408=-64.399,57.935,31.943,-152.8974,27.0473,0.0000
C01409=-61.254,61.254,31.948,-151.4856,25.5183,0.0000
C01410=-57.936,64.398,31.943,-150.1640,23.9390,0.0000
C01411=-54.626,67.259,31.951,-150.2002,23.7880,0.0000
C01412=-51.619,70.079,32.146,-152.4777,25.3540,0.0000
C01413=-50.255,72.374,32.633,-154.8677,26.4735,0.0000
C01414=-50.022,74.588,33.299,-157.0279,27.1227,0.0000
C01415=-50.362,76.980,33.980,-159.3588,27.4977,0.0000
C01416=-50.818,79.538,34.500,-162.2923,27.6007,0.0000
C01417=-50.816,82.144,34.757,-166.3861,27.1886,0.0000
C01418=-49.513,85.019,34.893,-172.0960,25.1202,0.0000
C01419=-47.019,87.765,35.004,-176.4080,21.3756,0.0000
C01420=-43.694,89.888,35.116,-178.7409,17.9455,0.0000
C01421=-40.099,91.601,35.190,-179.8842,15.3738,0.0000
C01422=-36.417,93.126,35.190,-168.9188,-10.7245,0.0000
C01423=-32.664,94.457,35.116,-166.2550,-11.7175,0.0000
C01424=-28.812,95.307,35.004,-162.1672,-12.5020,0.0000
C01425=-25.107,95.129,34.893,-156.5929,-12.2478,0.0000
C01426=-22.152,94.017,34.757,-151.4108,-10.0813,0.0000
C01427=-20.308,92.176,34.500,-148.4569,-7.8748,0.0000
C01428=-18.822,90.045,33.980,-146.5883,-6.0487,0.0000
C01429=-17.370,88.113,33.299,-145.2726,-4.4015,0.0000
C01430=-15.641,86.712,32.633,-144.2203,-2.6591,0.0000
C01431=-13.053,86.053,32.146,-143.2672,-0.4305,0.0000
C01432=-8.933,86.186,31.951,-142.6147,2.0827,0.0000
C01433=-4.570,86.503,31.943,-142.4957,1.9838,0.0000
C01434=0.000,86.627,31.948,-142.4647,0.0004,0.0000
C01435=0.000,85.325,33.722,-142.0369,0.0004,0.0000
C01436=4.451,85.206,33.716,-142.0680,-1.9932,0.0000
C01437=8.733,84.900,33.725,-142.1861,-1.9981,0.0000
C01438=12.808,84.808,33.943,-142.8511,0.6694,0.0000
C01439=15.338,85.570,34.490,-143.8100,2.9482,0.0000
C01440=17.019,87.137,35.239,-144.8677,4.7208,0.0000
C01441=18.435,89.289,36.009,-146.2129,6.4205,0.0000
C01442=19.887,91.675,36.600,-148.1683,8.3329,0.0000
C01443=21.692,93.766,36.894,-151.3315,10.6428,0.0000
C01444=24.671,95.076,37.049,-157.1379,12.9290,0.0000
C01445=28.465,95.370,37.176,-163.1840,12.8762,0.0000
C01446=32.445,94.529,37.304,-167.3718,11.7747,0.0000
C01447=36.342,93.155,37.389,-169.9560,10.6055,0.0000
C01448=40.172,91.569,37.389,179.4717,-14.5577,0.0000
C01449=43.901,89.784,37.304,-179.5776,-17.1955,0.0000
C01450=47.309,87.565,37.176,-177.4324,-20.9158,0.0000
C01451=49.784,84.674,37.049,-173.0456,-25.2119,0.0000
C01452=50.965,81.641,36.894,-166.7656,-27.6445,0.0000
C01453=50.762,78.886,36.600,-162.4082,-28.1308,0.0000
C01454=50.101,76.172,36.009,-159.3237,-28.0235,0.0000
C01455=49.580,73.649,35.239,-156.9183,-27.6282,0.0000
C01456=49.662,71.353,34.490,-154.7228,-26.9580,0.0000
C01457=50.912,69.025,33.943,-152.2841,-25.8010,0.0000
C01458=53.858,66.209,33.725,-149.8867,-24.1175,0.0000
C01459=57.102,63.397,33.716,-149.7877,-24.1936,0.0000
C01460=60.334,60.334,33.722,-151.1139,-25.7843,0.0000
C01461=63.397,57.102,33.716,-152.5296,-27.3228,0.0000
C01462=66.209,53.858,33.725,-152.6362,-27.2520,0.0000
C01463=69.025,50.912,33.943,-151.3611,-24.7537,0.0000
C01464=71.353,49.662,34.490,-150.6443,-22.3710,0.0000
C01465=73.649,49.580,35.239,-150.3620,-20.3250,0.0000
C01466=76.172,50.101,36.009,-150.3656,-18.1614,0.0000
C01467=78.886,50.762,36.600,-150.7133,-15.4583,0.0000
C01468=81.641,50.965,36.894,-151.7168,-11.7010,0.0000
C01469=84.674,49.784,37.049,-154.6247,-6.2891,0.0000
C01470=87.565,47.309,37.176,-159.0650,-2.3983,0.0000
C01471=89.784,43.901,37.304,-162.8041,-0.4035,0.0000
C01472=91.569,40.172,37.389,-165.4417,0.5113,0.0000
C01473=93.155,36.342,37.389,169.2333,-9.8707,0.0000
C01474=94.529,32.445,37.304,167.9418,-12.3583,0.0000
C01475=95.370,28.465,37.176,166.5690,-16.3810,0.0000
C01476=95.076,24.671,37.049,166.0104,-22.2510,0.0000
C01477=93.766,21.692,36.894,167.9114,-28.1310,0.0000
C01478=91.675,19.887,36.600,170.2184,-31.4569,0.0000
C01479=89.289,18.435,36.009,172.2892,-33.5470,0.0000
C01480=87.137,17.019,35.239,174.2340,-34.9957,0.0000
C01481=85.570,15.338,34.490,176.3487,-36.1345,0.0000
C01482=84.808,12.808,33.943,179.1602,-37.1460,0.0000
C01483=84.900,8.733,33.725,-177.4714,-37.7869,0.0000
C01484=85.206,4.451,33.716,-177.4736,-37.9050,0.0000
C01485=85.325,0.000,33.722,179.9995,-37.9631,0.0000
C01486=85.206,-4.451,33.716,177.4742,-37.9051,0.0000
C01487=84.900,-8.733,33.725,177.4725,-37.7868,0.0000
C01488=84.808,-12.808,33.943,-179.1598,-37.1459,0.0000
C01489=85.570,-15.338,34.490,-176.3490,-36.1345,0.0000
C01490=87.137,-17.019,35.239,-174.2344,-34.9957,0.0000
C01491=89.289,-18.435,36.009,-172.2896,-33.5471,0.0000
C01492=91.675,-19.887,36.600,-170.2187,-31.4571,0.0000
C01493=93.766,-21.692,36.894,-167.9116,-28.1311,0.0000
C01494=95.076,-24.671,37.049,-166.0104,-22.2510,0.0000
C01495=95.370,-28.465,37.176,-166.5690,-16.3810,0.0000
C01496=94.529,-32.445,37.304,-167.9418,-12.3583,0.0000
C01497=93.155,-36.342,37.389,-169.2333,-9.8707,0.0000
C01498=91.569,-40.172,37.389,165.4417,0.5113,0.0000
C01499=89.784,-43.901,37.304,162.8041,-0.4035,0.0000
C01500=87.565,-47.309,37.176,159.0650,-2.3983,0.0000
C01501=84.674,-49.784,37.049,154.6247,-6.2891,0.0000
C01502=81.641,-50.965,36.894,151.7167,-11.7008,0.0000
C01503=78.886,-50.762,36.600,150.7132,-15.4580,0.0000
C01504=76.172,-50.101,36.009,150.3654,-18.1611,0.0000
C01505=73.649,-49.580,35.239,150.3618,-20.3247,0.0000
C01506=71.353,-49.662,34.490,150.6441,-22.3708,0.0000
C01507=69.025,-50.912,33.943,151.3612,-24.7540,0.0000
C01508=66.209,-53.858,33.725,152.6368,-27.2528,0.0000
C01509=63.397,-57.102,33.716,152.5299,-27.3231,0.0000
C01510=60.334,-60.334,33.722,151.1134,-25.7837,0.0000
C01511=57.102,-63.397,33.716,149.7879,-24.1939,0.0000
C01512=53.858,-66.209,33.725,149.8874,-24.1181,0.0000
C01513=50.912,-69.025,33.943,152.2844,-25.8011,0.0000
C01514=49.662,-71.353,34.490,154.7227,-26.9579,0.0000
C01515=49.580,-73.649,35.239,156.9181,-27.6279,0.0000
C01516=50.101,-76.172,36.009,159.3234,-28.0233,0.0000
C01517=50.762,-78.886,36.600,162.4079,-28.1307,0.0000
C01518=50.965,-81.641,36.894,166.7654,-27.6445,0.0000
C01519=49.784,-84.674,37.049,173.0456,-25.2119,0.0000
C01520=47.309,-87.565,37.176,177.4324,-20.9158,0.0000
C01521=43.901,-89.784,37.304,179.5776,-17.1955,0.0000
C01522=40.172,-91.569,37.389,-179.4717,-14.5577,0.0000
C01523=36.342,-93.155,37.389,169.9560,10.6055,0.0000
C01524=32.445,-94.529,37.304,167.3718,11.7747,0.0000
C01525=28.465,-95.370,37.176,163.1840,12.8762,0.0000
C01526=24.671,-95.076,37.049,157.1379,12.9290,0.0000
C01527=21.692,-93.766,36.894,151.3315,10.6428,0.0000
C01528=19.887,-91.675,36.600,148.1683,8.3329,0.0000
C01529=18.435,-89.289,36.009,146.2129,6.4205,0.0000
C01530=17.019,-87.137,35.239,144.8677,4.7208,0.0000
C01531=15.338,-85.570,34.490,143.8100,2.9482,0.0000
C01532=12.808,-84.808,33.943,142.8511,0.6694,0.0000
C01533=8.733,-84.900,33.725,142.1861,-1.9981,0.0000
C01534=4.451,-85.206,33.716,142.0680,-1.9932,0.0000
C01535=0.000,-85.325,33.722,142.0369,0.0004,0.0000
C01536=0.000,-85.325,33.722,142.0369,0.0004,0.0000
C01537=-4.451,-85.206,33.716,142.0679,1.9927,0.0000
C01538=-8.733,-84.900,33.725,142.1862,1.9972,0.0000
C01539=-12.808,-84.808,33.943,142.8512,-0.6697,0.0000
C01540=-15.338,-85.570,34.490,143.8101,-2.9480,0.0000
C01541=-17.019,-87.137,35.239,144.8677,-4.7205,0.0000
C01542=-18.435,-89.289,36.009,146.2128,-6.4201,0.0000
C01543=-19.887,-91.675,36.600,148.1682,-8.3326,0.0000
C01544=-21.692,-93.766,36.894,151.3314,-10.6426,0.0000
C01545=-24.671,-95.076,37.049,157.1379,-12.9290,0.0000
C01546=-28.465,-95.370,37.176,163.1840,-12.8762,0.0000
C01547=-32.445,-94.529,37.304,167.3718,-11.7747,0.0000
C01548=-36.342,-93.155,37.389,169.9560,-10.6055,0.0000
C01549=-40.172,-91.569,37.389,-179.4717,14.5577,0.0000
C01550=-43.901,-89.784,37.304,179.5776,17.1955,0.0000
C01551=-47.309,-87.565,37.176,177.4324,20.9158,0.0000
C01552=-49.784,-84.674,37.049,173.0456,25.2119,0.0000
C01553=-50.965,-81.641,36.894,166.7656,27.6445,0.0000
C01554=-50.762,-78.886,36.600,162.4082,28.1308,0.0000
C01555=-50.101,-76.172,36.009,159.3237,28.0235,0.0000
C01556=-49.580,-73.649,35.239,156.9183,27.6282,0.0000
C01557=-49.662,-71.353,34.490,154.7228,26.9580,0.0000
C01558=-50.912,-69.025,33.943,152.2841,25.8010,0.0000
C01559=-53.858,-66.209,33.725,149.8867,24.1175,0.0000
C01560=-57.102,-63.397,33.716,149.7877,24.1936,0.0000
C01561=-60.334,-60.334,33.722,151.1139,25.7843,0.0000
C01562=-63.397,-57.102,33.716,152.5296,27.3228,0.0000
C01563=-66.209,-53.858,33.725,152.6362,27.2520,0.0000
C01564=-69.025,-50.912,33.943,151.3611,24.7537,0.0000
C01565=-71.353,-49.662,34.490,150.6443,22.3710,0.0000
C01566=-73.649,-49.580,35.239,150.3620,20.3250,0.0000
C01567=-76.172,-50.101,36.009,150.3656,18.1614,0.0000
C01568=-78.886,-50.762,36.600,150.7133,15.4583,0.0000
C01569=-81.641,-50.965,36.894,151.7168,11.7010,0.0000
C01570=-84.674,-49.784,37.049,154.6247,6.2891,0.0000
C01571=-87.565,-47.309,37.176,159.0650,2.3983,0.0000
C01572=-89.784,-43.901,37.304,162.8041,0.4035,0.0000
C01573=-91.569,-40.172,37.389,165.4417,-0.5113,0.0000
C01574=-93.155,-36.342,37.389,-169.2333,9.8707,0.0000
C01575=-94.529,-32.445,37.304,-167.9418,12.3583,0.0000
C01576=-95.370,-28.465,37.176,-166.5690,16.3810,0.0000
C01577=-95.076,-24.671,37.049,-166.0104,22.2510,0.0000
C01578=-93.766,-21.692,36.894,-167.9114,28.1310,0.0000
C01579=-91.675,-19.887,36.600,-170.2184,31.4569,0.0000
C01580=-89.289,-18.435,36.009,-172.2892,33.5470,0.0000
C01581=-87.137,-17.019,35.239,-174.2340,34.9957,0.0000
C01582=-85.570,-15.338,34.490,-176.3487,36.1345,0.0000
C01583=-84.808,-12.808,33.943,-179.1602,37.1460,0.0000
C01584=-84.900,-8.733,33.725,177.4714,37.7869,0.0000
C01585=-85.206,-4.451,33.716,177.4736,37.9050,0.0000
C01586=-85.325,0.000,33.722,-179.9995,37.9631,0.0000
C01587=-85.206,4.451,33.716,-177.4742,37.9051,0.0000
C01588=-84.900,8.733,33.725,-177.4725,37.7868,0.0000
C01589=-84.808,12.808,33.943,179.1598,37.1459,0.0000
C01590=-85.570,15.338,34.490,176.3490,36.1345,0.0000
C01591=-87.137,17.019,35.239,174.2344,34.9957,0.0000
C01592=-89.289,18.435,36.009,172.2896,33.5471,0.0000
C01593=-91.675,19.887,36.600,170.2187,31.4571,0.0000
C01594=-93.766,21.692,36.894,167.9116,28.1311,0.0000
C01595=-95.076,24.671,37.049,166.0104,22.2510,0.0000
C01596=-95.370,28.465,37.176,166.5690,16.3810,0.0000
C01597=-94.529,32.445,37.304,167.9418,12.3583,0.0000
C01598=-93.155,36.342,37.389,169.2333,9.8707,0.0000
C01599=-91.569,40.172,37.389,-165.4417,-0.5113,0.0000
C01600=-89.784,43.901,37.304,-162.8041,0.4035,0.0000
C01601=-87.565,47.309,37.176,-159.0650,2.3983,0.0000
C01602=-84.674,49.784,37.049,-154.6247,6.2891,0.0000
C01603=-81.641,50.965,36.894,-151.7167,11.7008,0.0000
C01604=-78.886,50.762,36.600,-150.7132,15.4580,0.0000
C01605=-76.172,50.101,36.009,-150.3654,18.1611,0.0000
C01606=-73.649,49.580,35.239,-150.3618,20.3247,0.0000
C01607=-71.353,49.662,34.490,-150.6441,22.3708,0.0000
C01608=-69.025,50.912,33.943,-151.3612,24.7540,0.0000
C01609=-66.209,53.858,33.725,-152.6368,27.2528,0.0000
C01610=-63.397,57.102,33.716,-152.5299,27.3231,0.0000
C01611=-60.334,60.334,33.722,-151.1134,25.7837,0.0000
C01612=-57.102,63.397,33.716,-149.7879,24.1939,0.0000
C01613=-53.858,66.209,33.725,-149.8874,24.1181,0.0000
C01614=-50.912,69.025,33.943,-152.2844,25.8011,0.0000
C01615=-49.662,71.353,34.490,-154.7227,26.9579,0.0000
C01616=-49.580,73.649,35.239,-156.9181,27.6279,0.0000
C01617=-50.101,76.172,36.009,-159.3234,28.0233,0.0000
C01618=-50.762,78.886,36.600,-162.4079,28.1307,0.0000
C01619=-50.965,81.641,36.894,-166.7654,27.6445,0.0000
C01620=-49.784,84.674,37.049,-173.0456,25.2119,0.0000
C01621=-47.309,87.565,37.176,-177.4324,20.9158,0.0000
C01622=-43.901,89.784,37.304,-179.5776,17.1955,0.0000
C01623=-40.172,91.569,37.389,179.4717,14.5577,0.0000
C01624=-36.342,93.155,37.389,-169.9560,-10.6055,0.0000
C01625=-32.445,94.529,37.304,-167.3718,-11.7747,0.0000
C01626=-28.465,95.370,37.176,-163.1840,-12.8762,0.0000
C01627=-24.671,95.076,37.049,-157.1379,-12.9290,0.0000
C01628=-21.692,93.766,36.894,-151.3314,-10.6426,0.0000
C01629=-19.887,91.675,36.600,-148.1682,-8.3326,0.0000
C01630=-18.435,89.289,36.009,-146.2128,-6.4201,0.0000
C01631=-17.019,87.137,35.239,-144.8677,-4.7205,0.0000
C01632=-15.338,85.570,34.490,-143.8101,-2.9480,0.0000
C01633=-12.808,84.808,33.943,-142.8512,-0.6697,0.0000
C01634=-8.733,84.900,33.725,-142.1862,1.9972,0.0000
C01635=-4.451,85.206,33.716,-142.0679,1.9927,0.0000
C01636=0.000,85.325,33.722,-142.0369,0.0004,0.0000
C01637=0.000,84.003,35.480,-141.6768,0.0003,0.0000
C01638=4.330,83.888,35.473,-141.7079,-1.9978,0.0000
C01639=8.530,83.594,35.484,-141.8255,-1.9113,0.0000
C01640=12.558,83.543,35.726,-142.5038,0.8975,0.0000
C01641=15.030,84.409,36.333,-143.4672,3.2159,0.0000
C01642=16.662,86.143,37.169,-144.5280,5.0137,0.0000
C01643=18.041,88.518,38.031,-145.9028,6.7672,0.0000
C01644=19.458,91.164,38.697,-147.9519,8.7720,0.0000
C01645=21.221,93.510,39.027,-151.3548,11.1943,0.0000
C01646=24.227,95.023,39.203,-157.8910,13.5428,0.0000
C01647=28.112,95.435,39.346,-164.4124,13.0755,0.0000
C01648=32.220,94.603,39.491,-168.6277,11.6199,0.0000
C01649=36.266,93.184,39.587,-171.0758,10.2870,0.0000
C01650=40.247,91.535,39.587,178.9188,-13.5446,0.0000
C01651=44.111,89.678,39.491,179.6508,-16.2003,0.0000
C01652=47.604,87.360,39.346,-178.4670,-20.1851,0.0000
C01653=50.060,84.322,39.203,-174.0956,-25.1075,0.0000
C01654=51.116,81.128,39.027,-167.2216,-28.0215,0.0000
C01655=50.704,78.221,38.697,-162.5706,-28.5979,0.0000
C01656=49.835,75.348,38.031,-159.3249,-28.4873,0.0000
C01657=49.130,72.694,37.169,-156.8445,-28.0709,0.0000
C01658=49.058,70.314,36.333,-154.6197,-27.3829,0.0000
C01659=50.194,67.954,35.726,-152.1415,-26.1962,0.0000
C01660=53.078,65.141,35.484,-149.6320,-24.4064,0.0000
C01661=56.256,62.380,35.473,-149.4718,-24.4096,0.0000
C01662=59.399,59.399,35.480,-150.7992,-26.0068,0.0000
C01663=62.380,56.256,35.473,-152.2169,-27.5520,0.0000
C01664=65.141,53.078,35.484,-152.2590,-27.4105,0.0000
C01665=67.954,50.194,35.726,-150.9052,-24.7896,0.0000
C01666=70.314,49.058,36.333,-150.1743,-22.3709,0.0000
C01667=72.694,49.130,37.169,-149.8854,-20.3024,0.0000
C01668=75.348,49.835,38.031,-149.8854,-18.0788,0.0000
C01669=78.221,50.704,38.697,-150.2563,-15.2478,0.0000
C01670=81.128,51.116,39.027,-151.3785,-11.2597,0.0000
C01671=84.322,50.060,39.203,-154.7752,-5.3448,0.0000
C01672=87.360,47.604,39.346,-159.8083,-1.4388,0.0000
C01673=89.678,44.111,39.491,-163.7994,0.3353,0.0000
C01674=91.535,40.247,39.587,-166.4530,1.0512,0.0000
C01675=93.184,36.266,39.587,169.5897,-8.7796,0.0000
C01676=94.603,32.220,39.491,168.1539,-11.1362,0.0000
C01677=95.435,28.112,39.346,166.4433,-15.1736,0.0000
C01678=95.023,24.227,39.203,165.4265,-21.4633,0.0000
C01679=93.510,21.221,39.027,167.2923,-28.0515,0.0000
C01680=91.164,19.458,38.697,169.6822,-31.6295,0.0000
C01681=88.518,18.041,38.031,171.8452,-33.8274,0.0000
C01682=86.143,16.662,37.169,173.8516,-35.3159,0.0000
C01683=84.409,15.030,36.333,176.0000,-36.4660,0.0000
C01684=83.543,12.558,35.726,178.8688,-37.4908,0.0000
C01685=83.594,8.530,35.484,-177.5693,-38.1494,0.0000
C01686=83.888,4.330,35.473,-177.4552,-38.2646,0.0000
C01687=84.003,0.000,35.480,179.9996,-38.3232,0.0000
C01688=83.888,-4.330,35.473,177.4557,-38.2647,0.0000
C01689=83.594,-8.530,35.484,177.5704,-38.1494,0.0000
C01690=83.543,-12.558,35.726,-178.8684,-37.4907,0.0000
C01691=84.409,-15.030,36.333,-176.0002,-36.4660,0.0000
C01692=86.143,-16.662,37.169,-173.8520,-35.3159,0.0000
C01693=88.518,-18.041,38.031,-171.8457,-33.8275,0.0000
C01694=91.164,-19.458,38.697,-169.6826,-31.6296,0.0000
C01695=93.510,-21.221,39.027,-167.2925,-28.0516,0.0000
C01696=95.023,-24.227,39.203,-165.4265,-21.4633,0.0000
C01697=95.435,-28.112,39.346,-166.4433,-15.1736,0.0000
C01698=94.603,-32.220,39.491,-168.1539,-11.1362,0.0000
C01699=93.184,-36.266,39.587,-169.5897,-8.7796,0.0000
C01700=91.535,-40.247,39.587,166.4530,1.0512,0.0000
C01701=89.678,-44.111,39.491,163.7994,0.3353,0.0000
C01702=87.360,-47.604,39.346,159.8083,-1.4388,0.0000
C01703=84.322,-50.060,39.203,154.7752,-5.3448,0.0000
C01704=81.128,-51.116,39.027,151.3785,-11.2595,0.0000
C01705=78.221,-50.704,38.697,150.2561,-15.2474,0.0000
C01706=75.348,-49.835,38.031,149.8852,-18.0785,0.0000
C01707=72.694,-49.130,37.169,149.8852,-20.3021,0.0000
C01708=70.314,-49.058,36.333,150.1741,-22.3707,0.0000
C01709=67.954,-50.194,35.726,150.9054,-24.7900,0.0000
C01710=65.141,-53.078,35.484,152.2596,-27.4112,0.0000
C01711=62.380,-56.256,35.473,152.2173,-27.5523,0.0000
C01712=59.399,-59.399,35.480,150.7988,-26.0063,0.0000
C01713=56.256,-62.380,35.473,149.4720,-24.4099,0.0000
C01714=53.078,-65.141,35.484,149.6327,-24.4071,0.0000
C01715=50.194,-67.954,35.726,152.1418,-26.1963,0.0000
C01716=49.058,-70.314,36.333,154.6196,-27.3827,0.0000
C01717=49.130,-72.694,37.169,156.8443,-28.0707,0.0000
C01718=49.835,-75.348,38.031,159.3246,-28.4871,0.0000
C01719=50.704,-78.221,38.697,162.5702,-28.5977,0.0000
C01720=51.116,-81.128,39.027,167.2214,-28.0214,0.0000
C01721=50.060,-84.322,39.203,174.0956,-25.1075,0.0000
C01722=47.604,-87.360,39.346,178.4670,-20.1851,0.0000
C01723=44.111,-89.678,39.491,-179.6508,-16.2003,0.0000
C01724=40.247,-91.535,39.587,-178.9188,-13.5446,0.0000
C01725=36.266,-93.184,39.587,171.0758,10.2870,0.0000
C01726=32.220,-94.603,39.491,168.6277,11.6199,0.0000
C01727=28.112,-95.435,39.346,164.4124,13.0755,0.0000
C01728=24.227,-95.023,39.203,157.8910,13.5428,0.0000
C01729=21.221,-93.510,39.027,151.3548,11.1943,0.0000
C01730=19.458,-91.164,38.697,147.9519,8.7720,0.0000
C01731=18.041,-88.518,38.031,145.9028,6.7672,0.0000
C01732=16.662,-86.143,37.169,144.5280,5.0137,0.0000
C01733=15.030,-84.409,36.333,143.4672,3.2159,0.0000
C01734=12.558,-83.543,35.726,142.5038,0.8975,0.0000
C01735=8.530,-83.594,35.484,141.8255,-1.9113,0.0000
C01736=4.330,-83.888,35.473,141.7079,-1.9978,0.0000
C01737=0.000,-84.003,35.480,141.6768,0.0003,0.0000
C01738=0.000,-84.003,35.480,141.6768,0.0003,0.0000
C01739=-4.330,-83.888,35.473,141.7078,1.9974,0.0000
C01740=-8.530,-83.594,35.484,141.8256,1.9104,0.0000
C01741=-12.558,-83.543,35.726,142.5039,-0.8979,0.0000
C01742=-15.030,-84.409,36.333,143.4672,-3.2157,0.0000
C01743=-16.662,-86.143,37.169,144.5280,-5.0134,0.0000
C01744=-18.041,-88.518,38.031,145.9027,-6.7668,0.0000
C01745=-19.458,-91.164,38.697,147.9518,-8.7716,0.0000
C01746=-21.221,-93.510,39.027,151.3546,-11.1941,0.0000
C01747=-24.227,-95.023,39.203,157.8910,-13.5428,0.0000
C01748=-28.112,-95.435,39.346,164.4124,-13.0755,0.0000
C01749=-32.220,-94.603,39.491,168.6277,-11.6199,0.0000
C01750=-36.266,-93.184,39.587,171.0758,-10.2870,0.0000
C01751=-40.247,-91.535,39.587,-178.9188,13.5446,0.0000
C01752=-44.111,-89.678,39.491,-179.6508,16.2003,0.0000
C01753=-47.604,-87.360,39.346,178.4670,20.1851,0.0000
C01754=-50.060,-84.322,39.203,174.0956,25.1075,0.0000
C01755=-51.116,-81.128,39.027,167.2216,28.0215,0.0000
C01756=-50.704,-78.221,38.697,162.5706,28.5979,0.0000
C01757=-49.835,-75.348,38.031,159.3249,28.4873,0.0000
C01758=-49.130,-72.694,37.169,156.8445,28.0709,0.0000
C01759=-49.058,-70.314,36.333,154.6197,27.3829,0.0000
C01760=-50.194,-67.954,35.726,152.1415,26.1962,0.0000
C01761=-53.078,-65.141,35.484,149.6320,24.4064,0.0000
C01762=-56.256,-62.380,35.473,149.4718,24.4096,0.0000
C01763=-59.399,-59.399,35.480,150.7992,26.0068,0.0000
C01764=-62.380,-56.256,35.473,152.2169,27.5520,0.0000
C01765=-65.141,-53.078,35.484,152.2590,27.4105,0.0000
C01766=-67.954,-50.194,35.726,150.9052,24.7896,0.0000
C01767=-70.314,-49.058,36.333,150.1743,22.3709,0.0000
C01768=-72.694,-49.130,37.169,149.8854,20.3024,0.0000
C01769=-75.348,-49.835,38.031,149.8854,18.0788,0.0000
C01770=-78.221,-50.704,38.697,150.2563,15.2478,0.0000
C01771=-81.128,-51.116,39.027,151.3785,11.2597,0.0000
C01772=-84.322,-50.060,39.203,154.7752,5.3448,0.0000
C01773=-87.360,-47.604,39.346,159.8083,1.4388,0.0000
C01774=-89.678,-44.111,39.491,163.7994,-0.3353,0.0000
C01775=-91.535,-40.247,39.587,166.4530,-1.0512,0.0000
C01776=-93.184,-36.266,39.587,-169.5897,8.7796,0.0000
C01777=-94.603,-32.220,39.491,-168.1539,11.1362,0.0000
C01778=-95.435,-28.112,39.346,-166.4433,15.1736,0.0000
C01779=-95.023,-24.227,39.203,-165.4265,21.4633,0.0000
C01780=-93.510,-21.221,39.027,-167.2923,28.0515,0.0000
C01781=-91.164,-19.458,38.697,-169.6822,31.6295,0.0000
C01782=-88.518,-18.041,38.031,-171.8452,33.8274,0.0000
C01783=-86.143,-16.662,37.169,-173.8516,35.3159,0.0000
C01784=-84.409,-15.030,36.333,-176.0000,36.4660,0.0000
C01785=-83.543,-12.558,35.726,-178.8688,37.4908,0.0000
C01786=-83.594,-8.530,35.484,177.5693,38.1494,0.0000
C01787=-83.888,-4.330,35.473,177.4552,38.2646,0.0000
C01788=-84.003,0.000,35.480,-179.9996,38.3232,0.0000
C01789=-83.888,4.330,35.473,-177.4557,38.2647,0.0000
C01790=-83.594,8.530,35.484,-177.5704,38.1494,0.0000
C01791=-83.543,12.558,35.726,178.8684,37.4907,0.0000
C01792=-84.409,15.030,36.333,176.0002,36.4660,0.0000
C01793=-86.143,16.662,37.169,173.8520,35.3159,0.0000
C01794=-88.518,18.041,38.031,171.8457,33.8275,0.0000
C01795=-91.164,19.458,38.697,169.6826,31.6296,0.0000
C01796=-93.510,21.221,39.027,167.2925,28.0516,0.0000
C01797=-95.023,24.227,39.203,165.4265,21.4633,0.0000
C01798=-95.435,28.112,39.346,166.4433,15.1736,0.0000
C01799=-94.603,32.220,39.491,168.1539,11.1362,0.0000
C01800=-93.184,36.266,39.587,169.5897,8.7796,0.0000
C01801=-91.535,40.247,39.587,-166.4530,-1.0512,0.0000
C01802=-89.678,44.111,39.491,-163.7994,-0.3353,0.0000
C01803=-87.360,47.604,39.346,-159.8083,1.4388,0.0000
C01804=-84.322,50.060,39.203,-154.7752,5.3448,0.0000
C01805=-81.128,51.116,39.027,-151.3785,11.2595,0.0000
C01806=-78.221,50.704,38.697,-150.2561,15.2474,0.0000
C01807=-75.348,49.835,38.031,-149.8852,18.0785,0.0000
C01808=-72.694,49.130,37.169,-149.8852,20.3021,0.0000
C01809=-70.314,49.058,36.333,-150.1741,22.3707,0.0000
C01810=-67.954,50.194,35.726,-150.9054,24.7900,0.0000
C01811=-65.141,53.078,35.484,-152.2596,27.4112,0.0000
C01812=-62.380,56.256,35.473,-152.2173,27.5523,0.0000
C01813=-59.399,59.399,35.480,-150.7988,26.0063,0.0000
C01814=-56.256,62.380,35.473,-149.4720,24.4099,0.0000
C01815=-53.078,65.141,35.484,-149.6327,24.4071,0.0000
C01816=-50.194,67.954,35.726,-152.1418,26.1963,0.0000
C01817=-49.058,70.314,36.333,-154.6196,27.3827,0.0000
C01818=-49.130,72.694,37.169,-156.8443,28.0707,0.0000
C01819=-49.835,75.348,38.031,-159.3246,28.4871,0.0000
C01820=-50.704,78.221,38.697,-162.5702,28.5977,0.0000
C01821=-51.116,81.128,39.027,-167.2214,28.0214,0.0000
C01822=-50.060,84.322,39.203,-174.0956,25.1075,0.0000
C01823=-47.604,87.360,39.346,-178.4670,20.1851,0.0000
C01824=-44.111,89.678,39.491,179.6508,16.2003,0.0000
C01825=-40.247,91.535,39.587,178.9188,13.5446,0.0000
C01826=-36.266,93.184,39.587,-171.0758,-10.2870,0.0000
C01827=-32.220,94.603,39.491,-168.6277,-11.6199,0.0000
C01828=-28.112,95.435,39.346,-164.4124,-13.0755,0.0000
C01829=-24.227,95.023,39.203,-157.8910,-13.5428,0.0000
C01830=-21.221,93.510,39.027,-151.3546,-11.1941,0.0000
C01831=-19.458,91.164,38.697,-147.9518,-8.7716,0.0000
C01832=-18.041,88.518,38.031,-145.9027,-6.7668,0.0000
C01833=-16.662,86.143,37.169,-144.5280,-5.0134,0.0000
C01834=-15.030,84.409,36.333,-143.4672,-3.2157,0.0000
C01835=-12.558,83.543,35.726,-142.5039,-0.8979,0.0000
C01836=-8.530,83.594,35.484,-141.8256,1.9104,0.0000
C01837=-4.330,83.888,35.473,-141.7078,1.9974,0.0000
C01838=0.000,84.003,35.480,-141.6768,0.0003,0.0000
C01839=0.000,82.662,37.225,-141.3795,0.0003,0.0000
C01840=4.208,82.553,37.217,-141.4105,-1.9985,0.0000
C01841=8.324,82.270,37.229,-141.5278,-1.8243,0.0000
C01842=12.305,82.260,37.495,-142.2197,1.1136,0.0000
C01843=14.718,83.232,38.165,-143.1858,3.4624,0.0000
C01844=16.299,85.134,39.090,-144.2478,5.2809,0.0000
C01845=17.640,87.735,40.048,-145.6523,7.0904,0.0000
C01846=19.021,90.644,40.789,-147.8040,9.1949,0.0000
C01847=20.743,93.250,41.159,-151.4856,11.7401,0.0000
C01848=23.775,94.968,41.355,-158.8727,14.0699,0.0000
C01849=27.752,95.500,41.515,-165.8427,13.0639,0.0000
C01850=31.992,94.679,41.678,-169.9901,11.2367,0.0000
C01851=36.189,93.214,41.785,-172.2431,9.7711,0.0000
C01852=40.323,91.502,41.785,178.4777,-12.3603,0.0000
C01853=44.326,89.570,41.678,178.9776,-14.9716,0.0000
C01854=47.905,87.153,41.515,-179.4760,-19.1659,0.0000
C01855=50.341,83.964,41.355,-175.2412,-24.7794,0.0000
C01856=51.270,80.606,41.159,-167.7610,-28.3185,0.0000
C01857=50.645,77.545,40.789,-162.7787,-29.0065,0.0000
C01858=49.565,74.511,40.048,-159.3591,-28.8940,0.0000
